LIN {X 0,Y 314.031,Z 449.566,A -85,B 0,C 180,E1 -15906.575,E2 -15906.575} C_VEL
LIN {X 0,Y 314.681,Z 456.551,A -85,B 0,C 180,E1 -15906.784,E2 -15906.784} C_VEL
LIN {X 0,Y 313.281,Z 518.504,A -85,B 0,C 180,E1 -15908.189,E2 -15908.189} C_VEL
LIN {X 0,Y 312.768,Z 530.956,A -85,B 0,C 180,E1 -15908.671,E2 -15908.671} C_VEL
LIN {X 0,Y 311.794,Z 543.197,A -85,B 0,C 180,E1 -15909.379,E2 -15909.379} C_VEL
LIN {X 0,Y 310.634,Z 555.216,A -85,B 0,C 180,E1 -15910.334,E2 -15910.334} C_VEL
LIN {X 0,Y 309.413,Z 566.12,A -85,B 0,C 180,E1 -15911.459,E2 -15911.459} C_VEL
LIN {X 0,Y 308.122,Z 576.138,A -85,B 0,C 180,E1 -15912.752,E2 -15912.752} C_VEL
LIN {X 0,Y 307.026,Z 586.271,A -85,B 0,C 180,E1 -15914.398,E2 -15914.398} C_VEL
LIN {X 0,Y 305.821,Z 596.058,A -85,B 0,C 180,E1 -15916.376,E2 -15916.376} C_VEL
LIN {X 0,Y 304.804,Z 603.833,A -85,B 0,C 180,E1 -15918.361,E2 -15918.361} C_VEL
LIN {X 0,Y 304.154,Z 610.997,A -85,B 0,C 180,E1 -15920.692,E2 -15920.692} C_VEL
LIN {X 0,Y 303.824,Z 615.751,A -85,B 0,C 180,E1 -15922.691,E2 -15922.691} C_VEL
LIN {X 0,Y 303.696,Z 619.372,A -85,B 0,C 180,E1 -15924.689,E2 -15924.689} C_VEL
LIN {X 0,Y 303.709,Z 621.23,A -85,B 0,C 180,E1 -15926.019,E2 -15926.019} C_VEL
LIN {X 0,Y 303.691,Z 622.612,A -85,B 0,C 180,E1 -15927.347,E2 -15927.347} C_VEL
LIN {X 0,Y 303.723,Z 623.593,A -85,B 0,C 180,E1 -15928.674,E2 -15928.674} C_VEL
LIN {X 0,Y 303.764,Z 624.179,A -85,B 0,C 180,E1 -15930,E2 -15930} C_VEL
LIN {X 0,Y 303.684,Z 624.356,A -85,B 0,C 180,E1 -15931.326,E2 -15931.326} C_VEL
LIN {X 0,Y 303.657,Z 624.102,A -85,B 0,C 180,E1 -15932.653,E2 -15932.653} C_VEL
LIN {X 0,Y 303.66,Z 623.46,A -85,B 0,C 180,E1 -15933.981,E2 -15933.981} C_VEL
LIN {X 0,Y 303.659,Z 622.155,A -85,B 0,C 180,E1 -15935.611,E2 -15935.611} C_VEL
LIN {X 0,Y 303.947,Z 619.106,A -85,B 0,C 180,E1 -15937.974,E2 -15937.974} C_VEL
LIN {X 0,Y 304.415,Z 615.463,A -85,B 0,C 180,E1 -15939.971,E2 -15939.971} C_VEL
LIN {X 0,Y 305.165,Z 610.729,A -85,B 0,C 180,E1 -15941.962,E2 -15941.962} C_VEL
LIN {X 0,Y 306.656,Z 603.648,A -85,B 0,C 180,E1 -15944.263,E2 -15944.263} C_VEL
LIN {X 0,Y 308.039,Z 596.351,A -85,B 0,C 180,E1 -15946.143,E2 -15946.143} C_VEL
LIN {X 0,Y 309.559,Z 588.201,A -85,B 0,C 180,E1 -15947.848,E2 -15947.848} C_VEL
LIN {X 0,Y 311.381,Z 578.704,A -85,B 0,C 180,E1 -15949.445,E2 -15949.445} C_VEL
LIN {X 0,Y 313.312,Z 568.196,A -85,B 0,C 180,E1 -15950.86,E2 -15950.86} C_VEL
LIN {X 0,Y 315.192,Z 556.51,A -85,B 0,C 180,E1 -15952.102,E2 -15952.102} C_VEL
LIN {X 0,Y 316.76,Z 545.154,A -85,B 0,C 180,E1 -15953.019,E2 -15953.019} C_VEL
LIN {X 0,Y 318.203,Z 531.649,A -85,B 0,C 180,E1 -15953.813,E2 -15953.813} C_VEL
LIN {X 0,Y 319.058,Z 519.098,A -85,B 0,C 180,E1 -15954.307,E2 -15954.307} C_VEL
LIN {X 0,Y 320.823,Z 456.805,A -85,B 0,C 180,E1 -15955.725,E2 -15955.725} C_VEL
LIN {X 0,Y 317.597,Z 436.667,A -85,B 0,C 180,E1 -15956.559,E2 -15956.559} C_VEL
LIN {X 0,Y 313.376,Z 415.766,A -85,B 0,C 180,E1 -15957.545,E2 -15957.545} C_VEL
LIN {X 0,Y 311.73,Z 410.591,A -85,B 0,C 180,E1 -15957.875,E2 -15957.875} C_VEL
LIN {X 0,Y 309.758,Z 401.062,A -85,B 0,C 180,E1 -15960.871,E2 -15960.871} C_VEL
LIN {X 0,Y 307.599,Z 391.784,A -85,B 0,C 180,E1 -15963.953,E2 -15963.953} C_VEL
LIN {X 0,Y 305.496,Z 383.432,A -85,B 0,C 180,E1 -15966.941,E2 -15966.941} C_VEL
LIN {X 0,Y 305.452,Z 383.433,A -85,B 0,C 180,E1 -15970.599,E2 -15970.599} C_VEL
LIN {X 0,Y 305.451,Z 383.431,A -85,B 0,C 180,E1 -15974.499,E2 -15974.499} C_VEL
LIN {X 0,Y 305.492,Z 383.426,A -85,B 0,C 180,E1 -15978.152,E2 -15978.152} C_VEL
LIN {X 0,Y 305.515,Z 383.425,A -85,B 0,C 180,E1 -15981.604,E2 -15981.604} C_VEL
LIN {X 0,Y 305.457,Z 383.433,A -85,B 0,C 180,E1 -15984.886,E2 -15984.886} C_VEL
LIN {X 0,Y 305.446,Z 383.436,A -85,B 0,C 180,E1 -15988.355,E2 -15988.355} C_VEL
LIN {X 0,Y 305.515,Z 383.428,A -85,B 0,C 180,E1 -15991.113,E2 -15991.113} C_VEL
LIN {X 0,Y 305.565,Z 383.4,A -85,B 0,C 180,E1 -15994.088,E2 -15994.088} C_VEL
LIN {X 0,Y 305.494,Z 383.43,A -85,B 0,C 180,E1 -15998.403,E2 -15998.403} C_VEL
LIN {X 0,Y 305.584,Z 383.414,A -85,B 0,C 180,E1 -16001.217,E2 -16001.217} C_VEL
LIN {X 0,Y 305.642,Z 383.406,A -85,B 0,C 180,E1 -16005.349,E2 -16005.349} C_VEL
LIN {X 0,Y 305.634,Z 383.406,A -85,B 0,C 180,E1 -16009.4,E2 -16009.4} C_VEL
LIN {X 0,Y 305.806,Z 383.391,A -85,B 0,C 180,E1 -16012.074,E2 -16012.074} C_VEL
LIN {X 0,Y 305.684,Z 383.399,A -85,B 0,C 180,E1 -16014.724,E2 -16014.724} C_VEL
LIN {X 0,Y 305.952,Z 383.366,A -85,B 0,C 180,E1 -16018.684,E2 -16018.684} C_VEL
LIN {X 0,Y 305.952,Z 383.374,A -85,B 0,C 180,E1 -16021.317,E2 -16021.317} C_VEL
LIN {X 0,Y 305.682,Z 383.408,A -85,B 0,C 180,E1 -16025.277,E2 -16025.277} C_VEL
LIN {X 0,Y 305.791,Z 383.386,A -85,B 0,C 180,E1 -16027.927,E2 -16027.927} C_VEL
LIN {X 0,Y 305.597,Z 383.414,A -85,B 0,C 180,E1 -16031.946,E2 -16031.946} C_VEL
LIN {X 0,Y 305.632,Z 383.414,A -85,B 0,C 180,E1 -16035.035,E2 -16035.035} C_VEL
LIN {X 0,Y 305.572,Z 383.42,A -85,B 0,C 180,E1 -16039.446,E2 -16039.446} C_VEL
LIN {X 0,Y 305.485,Z 383.432,A -85,B 0,C 180,E1 -16043.042,E2 -16043.042} C_VEL
LIN {X 0,Y 305.522,Z 383.403,A -85,B 0,C 180,E1 -16046.22,E2 -16046.22} C_VEL
LIN {X 0,Y 305.492,Z 383.431,A -85,B 0,C 180,E1 -16049.051,E2 -16049.051} C_VEL
LIN {X 0,Y 305.462,Z 383.435,A -85,B 0,C 180,E1 -16053.518,E2 -16053.518} C_VEL
LIN {X 0,Y 305.5,Z 383.429,A -85,B 0,C 180,E1 -16056.737,E2 -16056.737} C_VEL
LIN {X 0,Y 305.483,Z 383.437,A -85,B 0,C 180,E1 -16060.608,E2 -16060.608} C_VEL
LIN {X 0,Y 305.495,Z 383.433,A -85,B 0,C 180,E1 -16063.643,E2 -16063.643} C_VEL
LIN {X 0,Y 305.498,Z 383.436,A -85,B 0,C 180,E1 -16067.406,E2 -16067.406} C_VEL
LIN {X 0,Y 305.499,Z 383.524,A -85,B 0,C 180,E1 -16071.315,E2 -16071.315} C_VEL
LIN {X 0,Y 306.248,Z 386.681,A -85,B 0,C 180,E1 -16072.562,E2 -16072.562} C_VEL
LIN {X 0,Y 315.185,Z 404.698,A -85,B 0,C 180,E1 -16074.052,E2 -16074.052} C_VEL
LIN {X 0,Y 321.757,Z 419.845,A -85,B 0,C 180,E1 -16075.128,E2 -16075.128} C_VEL
LIN {X 0,Y 319.665,Z 493.003,A -85,B 0,C 180,E1 -16076.799,E2 -16076.799} C_VEL
LIN {X 0,Y 318.957,Z 504.93,A -85,B 0,C 180,E1 -16077.286,E2 -16077.286} C_VEL
LIN {X 0,Y 317.868,Z 517.514,A -85,B 0,C 180,E1 -16078.046,E2 -16078.046} C_VEL
LIN {X 0,Y 316.481,Z 528.377,A -85,B 0,C 180,E1 -16078.916,E2 -16078.916} C_VEL
LIN {X 0,Y 315.108,Z 539.273,A -85,B 0,C 180,E1 -16080.064,E2 -16080.064} C_VEL
LIN {X 0,Y 313.649,Z 548.685,A -85,B 0,C 180,E1 -16081.297,E2 -16081.297} C_VEL
LIN {X 0,Y 311.819,Z 558.321,A -85,B 0,C 180,E1 -16082.845,E2 -16082.845} C_VEL
LIN {X 0,Y 309.966,Z 567.861,A -85,B 0,C 180,E1 -16084.772,E2 -16084.772} C_VEL
LIN {X 0,Y 308.261,Z 575.922,A -85,B 0,C 180,E1 -16086.842,E2 -16086.842} C_VEL
LIN {X 0,Y 307.062,Z 581.197,A -85,B 0,C 180,E1 -16088.519,E2 -16088.519} C_VEL
LIN {X 0,Y 306.066,Z 585.733,A -85,B 0,C 180,E1 -16090.3,E2 -16090.3} C_VEL
LIN {X 0,Y 305.073,Z 590.158,A -85,B 0,C 180,E1 -16092.574,E2 -16092.574} C_VEL
LIN {X 0,Y 304.649,Z 592.146,A -85,B 0,C 180,E1 -16093.929,E2 -16093.929} C_VEL
LIN {X 0,Y 304.192,Z 594.355,A -85,B 0,C 180,E1 -16096.019,E2 -16096.019} C_VEL
LIN {X 0,Y 303.847,Z 595.527,A -85,B 0,C 180,E1 -16097.985,E2 -16097.985} C_VEL
LIN {X 0,Y 303.635,Z 595.748,A -85,B 0,C 180,E1 -16100.676,E2 -16100.676} C_VEL
LIN {X 0,Y 303.703,Z 595.242,A -85,B 0,C 180,E1 -16102.019,E2 -16102.019} C_VEL
LIN {X 0,Y 303.858,Z 593.743,A -85,B 0,C 180,E1 -16104.026,E2 -16104.026} C_VEL
LIN {X 0,Y 304.04,Z 590.269,A -85,B 0,C 180,E1 -16106.687,E2 -16106.687} C_VEL
LIN {X 0,Y 304.454,Z 586.504,A -85,B 0,C 180,E1 -16108.677,E2 -16108.677} C_VEL
LIN {X 0,Y 304.913,Z 581.638,A -85,B 0,C 180,E1 -16110.66,E2 -16110.66} C_VEL
LIN {X 0,Y 305.744,Z 575.501,A -85,B 0,C 180,E1 -16112.635,E2 -16112.635} C_VEL
LIN {X 0,Y 306.819,Z 567.863,A -85,B 0,C 180,E1 -16114.598,E2 -16114.598} C_VEL
LIN {X 0,Y 307.989,Z 558.298,A -85,B 0,C 180,E1 -16116.551,E2 -16116.551} C_VEL
LIN {X 0,Y 309.298,Z 548.412,A -85,B 0,C 180,E1 -16118.164,E2 -16118.164} C_VEL
LIN {X 0,Y 310.604,Z 537.252,A -85,B 0,C 180,E1 -16119.606,E2 -16119.606} C_VEL
LIN {X 0,Y 311.597,Z 526.36,A -85,B 0,C 180,E1 -16120.724,E2 -16120.724} C_VEL
LIN {X 0,Y 312.452,Z 515.426,A -85,B 0,C 180,E1 -16121.597,E2 -16121.597} C_VEL
LIN {X 0,Y 313.24,Z 502.643,A -85,B 0,C 180,E1 -16122.348,E2 -16122.348} C_VEL
LIN {X 0,Y 313.687,Z 490.148,A -85,B 0,C 180,E1 -16122.823,E2 -16122.823} C_VEL
LIN {X 0,Y 315.394,Z 413.357,A -85,B 0,C 180,E1 -16124.561,E2 -16124.561} C_VEL
LIN {X 0,Y 313.375,Z 405.881,A -85,B 0,C 180,E1 -16124.88,E2 -16124.88} C_VEL
LIN {X 0,Y 306.036,Z 385.635,A -85,B 0,C 180,E1 -16125.931,E2 -16125.931} C_VEL
LIN {X 0,Y 305.595,Z 383.422,A -85,B 0,C 180,E1 -16126.706,E2 -16126.706} C_VEL
LIN {X 0,Y 305.524,Z 383.429,A -85,B 0,C 180,E1 -16130.184,E2 -16130.184} C_VEL
LIN {X 0,Y 305.511,Z 383.428,A -85,B 0,C 180,E1 -16134.46,E2 -16134.46} C_VEL
LIN {X 0,Y 305.543,Z 383.423,A -85,B 0,C 180,E1 -16137.389,E2 -16137.389} C_VEL
LIN {X 0,Y 305.468,Z 383.437,A -85,B 0,C 180,E1 -16140.408,E2 -16140.408} C_VEL
LIN {X 0,Y 305.466,Z 383.435,A -85,B 0,C 180,E1 -16144.077,E2 -16144.077} C_VEL
LIN {X 0,Y 305.475,Z 383.433,A -85,B 0,C 180,E1 -16146.738,E2 -16146.738} C_VEL
LIN {X 0,Y 305.454,Z 383.433,A -85,B 0,C 180,E1 -16150.599,E2 -16150.599} C_VEL
LIN {X 0,Y 305.461,Z 383.435,A -85,B 0,C 180,E1 -16154.5,E2 -16154.5} C_VEL
LIN {X 0,Y 305.495,Z 383.427,A -85,B 0,C 180,E1 -16158.151,E2 -16158.151} C_VEL
LIN {X 0,Y 305.476,Z 383.427,A -85,B 0,C 180,E1 -16158.771,E2 -16158.771} C_VEL
LIN {X 0,Y 304.812,Z 383.515,A -85,B 0,C 180,E1 -16159.872,E2 -16159.872} C_VEL
LIN {X 0,Y 301.957,Z 383.87,A -85,B 0,C 180,E1 -16161.665,E2 -16161.665} C_VEL
LIN {X 0,Y 299.53,Z 384.171,A -85,B 0,C 180,E1 -16163.118,E2 -16163.118} C_VEL
LIN {X 0,Y 298.487,Z 384.3,A -85,B 0,C 180,E1 -16164.244,E2 -16164.244} C_VEL
LIN {X 0,Y 298.401,Z 384.306,A -85,B 0,C 180,E1 -16164.626,E2 -16164.626} C_VEL
LIN {X 0,Y 298.388,Z 384.315,A -85,B 0,C 180,E1 -16168.79,E2 -16168.79} C_VEL
LIN {X 0,Y 298.454,Z 384.307,A -85,B 0,C 180,E1 -16171.903,E2 -16171.903} C_VEL
LIN {X 0,Y 298.481,Z 384.297,A -85,B 0,C 180,E1 -16174.923,E2 -16174.923} C_VEL
LIN {X 0,Y 298.46,Z 384.305,A -85,B 0,C 180,E1 -16179.316,E2 -16179.316} C_VEL
LIN {X 0,Y 298.533,Z 384.296,A -85,B 0,C 180,E1 -16182.179,E2 -16182.179} C_VEL
LIN {X 0,Y 298.587,Z 384.282,A -85,B 0,C 180,E1 -16184.994,E2 -16184.994} C_VEL
LIN {X 0,Y 298.589,Z 384.288,A -85,B 0,C 180,E1 -16189.146,E2 -16189.146} C_VEL
LIN {X 0,Y 298.752,Z 384.27,A -85,B 0,C 180,E1 -16191.885,E2 -16191.885} C_VEL
LIN {X 0,Y 298.654,Z 384.273,A -85,B 0,C 180,E1 -16194.598,E2 -16194.598} C_VEL
LIN {X 0,Y 298.919,Z 384.248,A -85,B 0,C 180,E1 -16198.652,E2 -16198.652} C_VEL
LIN {X 0,Y 298.919,Z 384.248,A -85,B 0,C 180,E1 -16201.347,E2 -16201.347} C_VEL
LIN {X 0,Y 298.791,Z 384.264,A -85,B 0,C 180,E1 -16206.754,E2 -16206.754} C_VEL
LIN {X 0,Y 298.675,Z 384.278,A -85,B 0,C 180,E1 -16209.48,E2 -16209.48} C_VEL
LIN {X 0,Y 298.547,Z 384.295,A -85,B 0,C 180,E1 -16213.615,E2 -16213.615} C_VEL
LIN {X 0,Y 298.542,Z 384.297,A -85,B 0,C 180,E1 -16216.409,E2 -16216.409} C_VEL
LIN {X 0,Y 298.51,Z 384.299,A -85,B 0,C 180,E1 -16219.657,E2 -16219.657} C_VEL
LIN {X 0,Y 298.452,Z 384.307,A -85,B 0,C 180,E1 -16223.598,E2 -16223.598} C_VEL
LIN {X 0,Y 298.481,Z 384.303,A -85,B 0,C 180,E1 -16226.575,E2 -16226.575} C_VEL
LIN {X 0,Y 298.411,Z 384.314,A -85,B 0,C 180,E1 -16229.642,E2 -16229.642} C_VEL
LIN {X 0,Y 298.39,Z 384.314,A -85,B 0,C 180,E1 -16232.801,E2 -16232.801} C_VEL
LIN {X 0,Y 298.465,Z 384.305,A -85,B 0,C 180,E1 -16236.814,E2 -16236.814} C_VEL
LIN {X 0,Y 298.451,Z 384.307,A -85,B 0,C 180,E1 -16241.103,E2 -16241.103} C_VEL
LIN {X 0,Y 298.455,Z 384.306,A -85,B 0,C 180,E1 -16243.116,E2 -16243.116} C_VEL
LIN {X 0,Y 298.429,Z 384.309,A -85,B 0,C 180,E1 -16246.927,E2 -16246.927} C_VEL
LIN {X 0,Y 298.412,Z 384.312,A -85,B 0,C 180,E1 -16251.004,E2 -16251.004} C_VEL
LIN {X 0,Y 298.43,Z 384.313,A -85,B 0,C 180,E1 -16253.933,E2 -16253.933} C_VEL
LIN {X 0,Y 298.472,Z 384.46,A -85,B 0,C 180,E1 -16256.959,E2 -16256.959} C_VEL
LIN {X 0,Y 300.719,Z 394.722,A -85,B 0,C 180,E1 -16260.125,E2 -16260.125} C_VEL
LIN {X 0,Y 302.598,Z 404.683,A -85,B 0,C 180,E1 -16263.071,E2 -16263.071} C_VEL
LIN {X 0,Y 302.438,Z 408.558,A -85,B 0,C 180,E1 -16264.133,E2 -16264.133} C_VEL
LIN {X 0,Y 302.109,Z 410.992,A -85,B 0,C 180,E1 -16264.783,E2 -16264.783} C_VEL
LIN {X 0,Y 307.048,Z 447.973,A -85,B 0,C 180,E1 -16266.067,E2 -16266.067} C_VEL
LIN {X 0,Y 308.01,Z 456.583,A -85,B 0,C 180,E1 -16266.343,E2 -16266.343} C_VEL
LIN {X 0,Y 306.567,Z 518.379,A -85,B 0,C 180,E1 -16267.775,E2 -16267.775} C_VEL
LIN {X 0,Y 305.972,Z 531.497,A -85,B 0,C 180,E1 -16268.306,E2 -16268.306} C_VEL
LIN {X 0,Y 304.915,Z 544.079,A -85,B 0,C 180,E1 -16269.068,E2 -16269.068} C_VEL
LIN {X 0,Y 303.741,Z 555.836,A -85,B 0,C 180,E1 -16270.045,E2 -16270.045} C_VEL
LIN {X 0,Y 302.476,Z 566.54,A -85,B 0,C 180,E1 -16271.193,E2 -16271.193} C_VEL
LIN {X 0,Y 301.148,Z 576.39,A -85,B 0,C 180,E1 -16272.515,E2 -16272.515} C_VEL
LIN {X 0,Y 300.032,Z 586.208,A -85,B 0,C 180,E1 -16274.158,E2 -16274.158} C_VEL
LIN {X 0,Y 298.863,Z 595.373,A -85,B 0,C 180,E1 -16276.053,E2 -16276.053} C_VEL
LIN {X 0,Y 297.819,Z 603.237,A -85,B 0,C 180,E1 -16278.084,E2 -16278.084} C_VEL
LIN {X 0,Y 297.101,Z 610.45,A -85,B 0,C 180,E1 -16280.469,E2 -16280.469} C_VEL
LIN {X 0,Y 296.772,Z 615.252,A -85,B 0,C 180,E1 -16282.516,E2 -16282.516} C_VEL
LIN {X 0,Y 296.62,Z 618.915,A -85,B 0,C 180,E1 -16284.562,E2 -16284.562} C_VEL
LIN {X 0,Y 296.621,Z 620.803,A -85,B 0,C 180,E1 -16285.924,E2 -16285.924} C_VEL
LIN {X 0,Y 296.613,Z 622.214,A -85,B 0,C 180,E1 -16287.284,E2 -16287.284} C_VEL
LIN {X 0,Y 296.634,Z 623.213,A -85,B 0,C 180,E1 -16288.642,E2 -16288.642} C_VEL
LIN {X 0,Y 296.673,Z 623.818,A -85,B 0,C 180,E1 -16290,E2 -16290} C_VEL
LIN {X 0,Y 296.597,Z 624.023,A -85,B 0,C 180,E1 -16291.358,E2 -16291.358} C_VEL
LIN {X 0,Y 296.58,Z 623.796,A -85,B 0,C 180,E1 -16292.716,E2 -16292.716} C_VEL
LIN {X 0,Y 296.573,Z 623.172,A -85,B 0,C 180,E1 -16294.077,E2 -16294.077} C_VEL
LIN {X 0,Y 296.655,Z 620.753,A -85,B 0,C 180,E1 -16296.803,E2 -16296.803} C_VEL
LIN {X 0,Y 297.04,Z 617.811,A -85,B 0,C 180,E1 -16298.846,E2 -16298.846} C_VEL
LIN {X 0,Y 297.653,Z 613.853,A -85,B 0,C 180,E1 -16300.888,E2 -16300.888} C_VEL
LIN {X 0,Y 298.574,Z 608.782,A -85,B 0,C 180,E1 -16302.921,E2 -16302.921} C_VEL
LIN {X 0,Y 300.015,Z 602.442,A -85,B 0,C 180,E1 -16304.932,E2 -16304.932} C_VEL
LIN {X 0,Y 301.657,Z 594.115,A -85,B 0,C 180,E1 -16307.028,E2 -16307.028} C_VEL
LIN {X 0,Y 303.52,Z 584.719,A -85,B 0,C 180,E1 -16308.915,E2 -16308.915} C_VEL
LIN {X 0,Y 305.601,Z 574.521,A -85,B 0,C 180,E1 -16310.53,E2 -16310.53} C_VEL
LIN {X 0,Y 307.633,Z 563.029,A -85,B 0,C 180,E1 -16311.968,E2 -16311.968} C_VEL
LIN {X 0,Y 309.397,Z 551.737,A -85,B 0,C 180,E1 -16313.068,E2 -16313.068} C_VEL
LIN {X 0,Y 310.971,Z 540.209,A -85,B 0,C 180,E1 -16313.915,E2 -16313.915} C_VEL
LIN {X 0,Y 312.231,Z 527.003,A -85,B 0,C 180,E1 -16314.608,E2 -16314.608} C_VEL
LIN {X 0,Y 313.046,Z 514.207,A -85,B 0,C 180,E1 -16315.027,E2 -16315.027} C_VEL
LIN {X 0,Y 314.597,Z 457.765,A -85,B 0,C 180,E1 -16316.325,E2 -16316.325} C_VEL
LIN {X 0,Y 311.364,Z 437.492,A -85,B 0,C 180,E1 -16317.193,E2 -16317.193} C_VEL
LIN {X 0,Y 307.278,Z 417.254,A -85,B 0,C 180,E1 -16318.181,E2 -16318.181} C_VEL
LIN {X 0,Y 304.522,Z 410.161,A -85,B 0,C 180,E1 -16318.718,E2 -16318.718} C_VEL
LIN {X 0,Y 302.101,Z 399.117,A -85,B 0,C 180,E1 -16322.348,E2 -16322.348} C_VEL
LIN {X 0,Y 299.654,Z 389.019,A -85,B 0,C 180,E1 -16325.897,E2 -16325.897} C_VEL
LIN {X 0,Y 298.473,Z 384.306,A -85,B 0,C 180,E1 -16327.683,E2 -16327.683} C_VEL
LIN {X 0,Y 298.383,Z 384.314,A -85,B 0,C 180,E1 -16331.261,E2 -16331.261} C_VEL
LIN {X 0,Y 298.413,Z 384.308,A -85,B 0,C 180,E1 -16335.046,E2 -16335.046} C_VEL
LIN {X 0,Y 298.451,Z 384.302,A -85,B 0,C 180,E1 -16338.75,E2 -16338.75} C_VEL
LIN {X 0,Y 298.443,Z 384.305,A -85,B 0,C 180,E1 -16342.246,E2 -16342.246} C_VEL
LIN {X 0,Y 298.403,Z 384.314,A -85,B 0,C 180,E1 -16345.581,E2 -16345.581} C_VEL
LIN {X 0,Y 298.39,Z 384.316,A -85,B 0,C 180,E1 -16348.791,E2 -16348.791} C_VEL
LIN {X 0,Y 298.458,Z 384.307,A -85,B 0,C 180,E1 -16351.904,E2 -16351.904} C_VEL
LIN {X 0,Y 298.479,Z 384.277,A -85,B 0,C 180,E1 -16354.924,E2 -16354.924} C_VEL
LIN {X 0,Y 298.444,Z 384.309,A -85,B 0,C 180,E1 -16359.315,E2 -16359.315} C_VEL
LIN {X 0,Y 298.531,Z 384.296,A -85,B 0,C 180,E1 -16362.179,E2 -16362.179} C_VEL
LIN {X 0,Y 298.587,Z 384.284,A -85,B 0,C 180,E1 -16364.995,E2 -16364.995} C_VEL
LIN {X 0,Y 298.589,Z 384.284,A -85,B 0,C 180,E1 -16369.147,E2 -16369.147} C_VEL
LIN {X 0,Y 298.751,Z 384.27,A -85,B 0,C 180,E1 -16371.886,E2 -16371.886} C_VEL
LIN {X 0,Y 298.655,Z 384.274,A -85,B 0,C 180,E1 -16374.599,E2 -16374.599} C_VEL
LIN {X 0,Y 298.919,Z 384.242,A -85,B 0,C 180,E1 -16378.653,E2 -16378.653} C_VEL
LIN {X 0,Y 298.919,Z 384.25,A -85,B 0,C 180,E1 -16381.348,E2 -16381.348} C_VEL
LIN {X 0,Y 298.781,Z 384.265,A -85,B 0,C 180,E1 -16386.755,E2 -16386.755} C_VEL
LIN {X 0,Y 298.629,Z 384.284,A -85,B 0,C 180,E1 -16389.483,E2 -16389.483} C_VEL
LIN {X 0,Y 298.546,Z 384.293,A -85,B 0,C 180,E1 -16393.616,E2 -16393.616} C_VEL
LIN {X 0,Y 298.543,Z 384.292,A -85,B 0,C 180,E1 -16396.409,E2 -16396.409} C_VEL
LIN {X 0,Y 298.507,Z 384.301,A -85,B 0,C 180,E1 -16399.655,E2 -16399.655} C_VEL
LIN {X 0,Y 298.453,Z 384.307,A -85,B 0,C 180,E1 -16403.599,E2 -16403.599} C_VEL
LIN {X 0,Y 298.481,Z 384.279,A -85,B 0,C 180,E1 -16406.576,E2 -16406.576} C_VEL
LIN {X 0,Y 298.417,Z 384.313,A -85,B 0,C 180,E1 -16409.642,E2 -16409.642} C_VEL
LIN {X 0,Y 298.392,Z 384.316,A -85,B 0,C 180,E1 -16412.801,E2 -16412.801} C_VEL
LIN {X 0,Y 298.468,Z 384.305,A -85,B 0,C 180,E1 -16416.815,E2 -16416.815} C_VEL
LIN {X 0,Y 298.45,Z 384.31,A -85,B 0,C 180,E1 -16421.251,E2 -16421.251} C_VEL
LIN {X 0,Y 298.417,Z 384.319,A -85,B 0,C 180,E1 -16425.048,E2 -16425.048} C_VEL
LIN {X 0,Y 298.42,Z 384.318,A -85,B 0,C 180,E1 -16428.746,E2 -16428.746} C_VEL
LIN {X 0,Y 298.442,Z 384.336,A -85,B 0,C 180,E1 -16430.593,E2 -16430.593} C_VEL
LIN {X 0,Y 299.127,Z 387.198,A -85,B 0,C 180,E1 -16431.71,E2 -16431.71} C_VEL
LIN {X 0,Y 308.479,Z 405.641,A -85,B 0,C 180,E1 -16433.333,E2 -16433.333} C_VEL
LIN {X 0,Y 315.617,Z 421.901,A -85,B 0,C 180,E1 -16434.544,E2 -16434.544} C_VEL
LIN {X 0,Y 313.411,Z 493.482,A -85,B 0,C 180,E1 -16436.204,E2 -16436.204} C_VEL
LIN {X 0,Y 312.64,Z 505.613,A -85,B 0,C 180,E1 -16436.711,E2 -16436.711} C_VEL
LIN {X 0,Y 311.491,Z 518.351,A -85,B 0,C 180,E1 -16437.503,E2 -16437.503} C_VEL
LIN {X 0,Y 310.045,Z 529.099,A -85,B 0,C 180,E1 -16438.387,E2 -16438.387} C_VEL
LIN {X 0,Y 308.6,Z 539.894,A -85,B 0,C 180,E1 -16439.555,E2 -16439.555} C_VEL
LIN {X 0,Y 306.869,Z 550.302,A -85,B 0,C 180,E1 -16440.971,E2 -16440.971} C_VEL
LIN {X 0,Y 304.992,Z 559.748,A -85,B 0,C 180,E1 -16442.558,E2 -16442.558} C_VEL
LIN {X 0,Y 303.095,Z 568.961,A -85,B 0,C 180,E1 -16444.497,E2 -16444.497} C_VEL
LIN {X 0,Y 301.294,Z 576.936,A -85,B 0,C 180,E1 -16446.638,E2 -16446.638} C_VEL
LIN {X 0,Y 299.845,Z 582.994,A -85,B 0,C 180,E1 -16448.697,E2 -16448.697} C_VEL
LIN {X 0,Y 298.742,Z 587.747,A -85,B 0,C 180,E1 -16450.771,E2 -16450.771} C_VEL
LIN {X 0,Y 297.913,Z 591.348,A -85,B 0,C 180,E1 -16452.85,E2 -16452.85} C_VEL
LIN {X 0,Y 297.318,Z 593.901,A -85,B 0,C 180,E1 -16454.929,E2 -16454.929} C_VEL
LIN {X 0,Y 297.053,Z 595.084,A -85,B 0,C 180,E1 -16456.315,E2 -16456.315} C_VEL
LIN {X 0,Y 296.821,Z 595.816,A -85,B 0,C 180,E1 -16457.696,E2 -16457.696} C_VEL
LIN {X 0,Y 296.541,Z 596.101,A -85,B 0,C 180,E1 -16460.451,E2 -16460.451} C_VEL
LIN {X 0,Y 296.606,Z 595.653,A -85,B 0,C 180,E1 -16461.827,E2 -16461.827} C_VEL
LIN {X 0,Y 296.765,Z 594.02,A -85,B 0,C 180,E1 -16464.074,E2 -16464.074} C_VEL
LIN {X 0,Y 296.946,Z 590.813,A -85,B 0,C 180,E1 -16466.608,E2 -16466.608} C_VEL
LIN {X 0,Y 297.375,Z 587.117,A -85,B 0,C 180,E1 -16468.646,E2 -16468.646} C_VEL
LIN {X 0,Y 297.836,Z 582.328,A -85,B 0,C 180,E1 -16470.676,E2 -16470.676} C_VEL
LIN {X 0,Y 298.671,Z 576.275,A -85,B 0,C 180,E1 -16472.697,E2 -16472.697} C_VEL
LIN {X 0,Y 299.766,Z 568.755,A -85,B 0,C 180,E1 -16474.707,E2 -16474.707} C_VEL
LIN {X 0,Y 300.757,Z 561.086,A -85,B 0,C 180,E1 -16476.373,E2 -16476.373} C_VEL
LIN {X 0,Y 302.145,Z 550.656,A -85,B 0,C 180,E1 -16478.191,E2 -16478.191} C_VEL
LIN {X 0,Y 303.46,Z 540.042,A -85,B 0,C 180,E1 -16479.666,E2 -16479.666} C_VEL
LIN {X 0,Y 304.53,Z 529.786,A -85,B 0,C 180,E1 -16480.807,E2 -16480.807} C_VEL
LIN {X 0,Y 305.535,Z 517.548,A -85,B 0,C 180,E1 -16481.863,E2 -16481.863} C_VEL
LIN {X 0,Y 306.434,Z 504.645,A -85,B 0,C 180,E1 -16482.668,E2 -16482.668} C_VEL
LIN {X 0,Y 306.928,Z 492.158,A -85,B 0,C 180,E1 -16483.195,E2 -16483.195} C_VEL
LIN {X 0,Y 308.756,Z 414.425,A -85,B 0,C 180,E1 -16484.997,E2 -16484.997} C_VEL
LIN {X 0,Y 305.841,Z 404.808,A -85,B 0,C 180,E1 -16485.445,E2 -16485.445} C_VEL
LIN {X 0,Y 298.882,Z 385.947,A -85,B 0,C 180,E1 -16486.477,E2 -16486.477} C_VEL
LIN {X 0,Y 298.535,Z 384.299,A -85,B 0,C 180,E1 -16487.113,E2 -16487.113} C_VEL
LIN {X 0,Y 298.455,Z 384.31,A -85,B 0,C 180,E1 -16490.684,E2 -16490.684} C_VEL
LIN {X 0,Y 298.489,Z 384.297,A -85,B 0,C 180,E1 -16495.075,E2 -16495.075} C_VEL
LIN {X 0,Y 298.478,Z 384.305,A -85,B 0,C 180,E1 -16498.093,E2 -16498.093} C_VEL
LIN {X 0,Y 298.397,Z 384.315,A -85,B 0,C 180,E1 -16502.799,E2 -16502.799} C_VEL
LIN {X 0,Y 298.447,Z 384.308,A -85,B 0,C 180,E1 -16506.807,E2 -16506.807} C_VEL
LIN {X 0,Y 298.409,Z 384.311,A -85,B 0,C 180,E1 -16509.485,E2 -16509.485} C_VEL
LIN {X 0,Y 298.425,Z 384.309,A -85,B 0,C 180,E1 -16513.108,E2 -16513.108} C_VEL
LIN {X 0,Y 298.466,Z 384.299,A -85,B 0,C 180,E1 -16516.931,E2 -16516.931} C_VEL
LIN {X 0,Y 298.438,Z 384.308,A -85,B 0,C 180,E1 -16520.997,E2 -16520.997} C_VEL
LIN {X 0,Y 298.401,Z 384.306,A -85,B 0,C 180,E1 -16524.626,E2 -16524.626} C_VEL
LIN {X 0,Y 297.734,Z 384.39,A -85,B 0,C 180,E1 -16525.752,E2 -16525.752} C_VEL
LIN {X 0,Y 294.897,Z 384.748,A -85,B 0,C 180,E1 -16527.585,E2 -16527.585} C_VEL
LIN {X 0,Y 292.49,Z 385.054,A -85,B 0,C 180,E1 -16529.073,E2 -16529.073} C_VEL
LIN {X 0,Y 291.455,Z 385.182,A -85,B 0,C 180,E1 -16530.225,E2 -16530.225} C_VEL
LIN {X 0,Y 291.368,Z 385.19,A -85,B 0,C 180,E1 -16530.616,E2 -16530.616} C_VEL
LIN {X 0,Y 291.41,Z 385.179,A -85,B 0,C 180,E1 -16534.271,E2 -16534.271} C_VEL
LIN {X 0,Y 291.385,Z 385.185,A -85,B 0,C 180,E1 -16537.299,E2 -16537.299} C_VEL
LIN {X 0,Y 291.458,Z 385.18,A -85,B 0,C 180,E1 -16540.27,E2 -16540.27} C_VEL
LIN {X 0,Y 291.535,Z 385.161,A -85,B 0,C 180,E1 -16544.634,E2 -16544.634} C_VEL
LIN {X 0,Y 291.533,Z 385.168,A -85,B 0,C 180,E1 -16548.88,E2 -16548.88} C_VEL
LIN {X 0,Y 291.703,Z 385.147,A -85,B 0,C 180,E1 -16551.688,E2 -16551.688} C_VEL
LIN {X 0,Y 291.625,Z 385.148,A -85,B 0,C 180,E1 -16554.468,E2 -16554.468} C_VEL
LIN {X 0,Y 291.885,Z 385.124,A -85,B 0,C 180,E1 -16558.62,E2 -16558.62} C_VEL
LIN {X 0,Y 291.885,Z 385.124,A -85,B 0,C 180,E1 -16561.379,E2 -16561.379} C_VEL
LIN {X 0,Y 291.74,Z 385.141,A -85,B 0,C 180,E1 -16566.918,E2 -16566.918} C_VEL
LIN {X 0,Y 291.623,Z 385.157,A -85,B 0,C 180,E1 -16569.712,E2 -16569.712} C_VEL
LIN {X 0,Y 291.516,Z 385.172,A -85,B 0,C 180,E1 -16573.95,E2 -16573.95} C_VEL
LIN {X 0,Y 291.481,Z 385.174,A -85,B 0,C 180,E1 -16576.818,E2 -16576.818} C_VEL
LIN {X 0,Y 291.446,Z 385.181,A -85,B 0,C 180,E1 -16579.875,E2 -16579.875} C_VEL
LIN {X 0,Y 291.394,Z 385.189,A -85,B 0,C 180,E1 -16584.206,E2 -16584.206} C_VEL
LIN {X 0,Y 291.414,Z 385.183,A -85,B 0,C 180,E1 -16587.272,E2 -16587.272} C_VEL
LIN {X 0,Y 291.328,Z 385.195,A -85,B 0,C 180,E1 -16590.438,E2 -16590.438} C_VEL
LIN {X 0,Y 291.339,Z 385.196,A -85,B 0,C 180,E1 -16593.699,E2 -16593.699} C_VEL
LIN {X 0,Y 291.4,Z 385.185,A -85,B 0,C 180,E1 -16597.262,E2 -16597.262} C_VEL
LIN {X 0,Y 291.401,Z 385.185,A -85,B 0,C 180,E1 -16600.631,E2 -16600.631} C_VEL
LIN {X 0,Y 291.349,Z 385.191,A -85,B 0,C 180,E1 -16604.39,E2 -16604.39} C_VEL
LIN {X 0,Y 291.35,Z 385.193,A -85,B 0,C 180,E1 -16608.399,E2 -16608.399} C_VEL
LIN {X 0,Y 291.362,Z 385.191,A -85,B 0,C 180,E1 -16611.161,E2 -16611.161} C_VEL
LIN {X 0,Y 291.383,Z 385.19,A -85,B 0,C 180,E1 -16614.63,E2 -16614.63} C_VEL
LIN {X 0,Y 291.431,Z 385.378,A -85,B 0,C 180,E1 -16616.545,E2 -16616.545} C_VEL
LIN {X 0,Y 293.965,Z 397.107,A -85,B 0,C 180,E1 -16620.26,E2 -16620.26} C_VEL
LIN {X 0,Y 295.562,Z 405.409,A -85,B 0,C 180,E1 -16622.776,E2 -16622.776} C_VEL
LIN {X 0,Y 295.707,Z 408.051,A -85,B 0,C 180,E1 -16623.537,E2 -16623.537} C_VEL
LIN {X 0,Y 295.332,Z 410.69,A -85,B 0,C 180,E1 -16624.259,E2 -16624.259} C_VEL
LIN {X 0,Y 300.207,Z 447.289,A -85,B 0,C 180,E1 -16625.567,E2 -16625.567} C_VEL
LIN {X 0,Y 301.35,Z 457.164,A -85,B 0,C 180,E1 -16625.896,E2 -16625.896} C_VEL
LIN {X 0,Y 299.869,Z 518.251,A -85,B 0,C 180,E1 -16627.342,E2 -16627.342} C_VEL
LIN {X 0,Y 299.248,Z 531.269,A -85,B 0,C 180,E1 -16627.883,E2 -16627.883} C_VEL
LIN {X 0,Y 298.157,Z 543.824,A -85,B 0,C 180,E1 -16628.662,E2 -16628.662} C_VEL
LIN {X 0,Y 296.854,Z 556.433,A -85,B 0,C 180,E1 -16629.743,E2 -16629.743} C_VEL
LIN {X 0,Y 295.327,Z 568.21,A -85,B 0,C 180,E1 -16631.081,E2 -16631.081} C_VEL
LIN {X 0,Y 293.914,Z 578.799,A -85,B 0,C 180,E1 -16632.609,E2 -16632.609} C_VEL
LIN {X 0,Y 292.942,Z 587.189,A -85,B 0,C 180,E1 -16634.108,E2 -16634.108} C_VEL
LIN {X 0,Y 291.741,Z 596.151,A -85,B 0,C 180,E1 -16636.061,E2 -16636.061} C_VEL
LIN {X 0,Y 290.68,Z 603.771,A -85,B 0,C 180,E1 -16638.141,E2 -16638.141} C_VEL
LIN {X 0,Y 290.065,Z 609.903,A -85,B 0,C 180,E1 -16640.235,E2 -16640.235} C_VEL
LIN {X 0,Y 289.7,Z 614.75,A -85,B 0,C 180,E1 -16642.332,E2 -16642.332} C_VEL
LIN {X 0,Y 289.556,Z 618.458,A -85,B 0,C 180,E1 -16644.429,E2 -16644.429} C_VEL
LIN {X 0,Y 289.537,Z 620.369,A -85,B 0,C 180,E1 -16645.824,E2 -16645.824} C_VEL
LIN {X 0,Y 289.538,Z 621.816,A -85,B 0,C 180,E1 -16647.217,E2 -16647.217} C_VEL
LIN {X 0,Y 289.548,Z 622.833,A -85,B 0,C 180,E1 -16648.609,E2 -16648.609} C_VEL
LIN {X 0,Y 289.583,Z 623.456,A -85,B 0,C 180,E1 -16650,E2 -16650} C_VEL
LIN {X 0,Y 289.512,Z 623.683,A -85,B 0,C 180,E1 -16651.391,E2 -16651.391} C_VEL
LIN {X 0,Y 289.505,Z 623.49,A -85,B 0,C 180,E1 -16652.783,E2 -16652.783} C_VEL
LIN {X 0,Y 289.48,Z 621.949,A -85,B 0,C 180,E1 -16655.499,E2 -16655.499} C_VEL
LIN {X 0,Y 289.581,Z 620.502,A -85,B 0,C 180,E1 -16656.97,E2 -16656.97} C_VEL
LIN {X 0,Y 290.006,Z 617.599,A -85,B 0,C 180,E1 -16659.063,E2 -16659.063} C_VEL
LIN {X 0,Y 290.643,Z 613.682,A -85,B 0,C 180,E1 -16661.154,E2 -16661.154} C_VEL
LIN {X 0,Y 291.639,Z 608.656,A -85,B 0,C 180,E1 -16663.234,E2 -16663.234} C_VEL
LIN {X 0,Y 293.128,Z 602.375,A -85,B 0,C 180,E1 -16665.291,E2 -16665.291} C_VEL
LIN {X 0,Y 294.754,Z 594.672,A -85,B 0,C 180,E1 -16667.31,E2 -16667.31} C_VEL
LIN {X 0,Y 296.411,Z 586.589,A -85,B 0,C 180,E1 -16669.027,E2 -16669.027} C_VEL
LIN {X 0,Y 298.513,Z 576.905,A -85,B 0,C 180,E1 -16670.68,E2 -16670.68} C_VEL
LIN {X 0,Y 300.639,Z 566.169,A -85,B 0,C 180,E1 -16672.144,E2 -16672.144} C_VEL
LIN {X 0,Y 302.456,Z 555.753,A -85,B 0,C 180,E1 -16673.267,E2 -16673.267} C_VEL
LIN {X 0,Y 304.104,Z 544.377,A -85,B 0,C 180,E1 -16674.218,E2 -16674.218} C_VEL
LIN {X 0,Y 305.543,Z 531.604,A -85,B 0,C 180,E1 -16675.002,E2 -16675.002} C_VEL
LIN {X 0,Y 306.569,Z 518.21,A -85,B 0,C 180,E1 -16675.548,E2 -16675.548} C_VEL
LIN {X 0,Y 308.41,Z 458.561,A -85,B 0,C 180,E1 -16676.955,E2 -16676.955} C_VEL
LIN {X 0,Y 305.24,Z 438.655,A -85,B 0,C 180,E1 -16677.835,E2 -16677.835} C_VEL
LIN {X 0,Y 301.365,Z 419.447,A -85,B 0,C 180,E1 -16678.807,E2 -16678.807} C_VEL
LIN {X 0,Y 298.357,Z 412.643,A -85,B 0,C 180,E1 -16679.359,E2 -16679.359} C_VEL
LIN {X 0,Y 297.245,Z 409.759,A -85,B 0,C 180,E1 -16679.603,E2 -16679.603} C_VEL
LIN {X 0,Y 294.921,Z 399.119,A -85,B 0,C 180,E1 -16683.235,E2 -16683.235} C_VEL
LIN {X 0,Y 292.384,Z 389.052,A -85,B 0,C 180,E1 -16686.935,E2 -16686.935} C_VEL
LIN {X 0,Y 291.372,Z 385.189,A -85,B 0,C 180,E1 -16688.432,E2 -16688.432} C_VEL
LIN {X 0,Y 291.337,Z 385.191,A -85,B 0,C 180,E1 -16692.488,E2 -16692.488} C_VEL
LIN {X 0,Y 291.367,Z 385.186,A -85,B 0,C 180,E1 -16696.353,E2 -16696.353} C_VEL
LIN {X 0,Y 291.409,Z 385.181,A -85,B 0,C 180,E1 -16700.51,E2 -16700.51} C_VEL
LIN {X 0,Y 291.429,Z 385.178,A -85,B 0,C 180,E1 -16702.923,E2 -16702.923} C_VEL
LIN {X 0,Y 291.34,Z 385.193,A -85,B 0,C 180,E1 -16706.301,E2 -16706.301} C_VEL
LIN {X 0,Y 291.382,Z 385.185,A -85,B 0,C 180,E1 -16710.26,E2 -16710.26} C_VEL
LIN {X 0,Y 291.41,Z 385.16,A -85,B 0,C 180,E1 -16714.272,E2 -16714.272} C_VEL
LIN {X 0,Y 291.376,Z 385.18,A -85,B 0,C 180,E1 -16717.299,E2 -16717.299} C_VEL
LIN {X 0,Y 291.452,Z 385.175,A -85,B 0,C 180,E1 -16720.27,E2 -16720.27} C_VEL
LIN {X 0,Y 291.534,Z 385.163,A -85,B 0,C 180,E1 -16724.634,E2 -16724.634} C_VEL
LIN {X 0,Y 291.532,Z 385.164,A -85,B 0,C 180,E1 -16728.881,E2 -16728.881} C_VEL
LIN {X 0,Y 291.702,Z 385.149,A -85,B 0,C 180,E1 -16731.689,E2 -16731.689} C_VEL
LIN {X 0,Y 291.625,Z 385.149,A -85,B 0,C 180,E1 -16734.469,E2 -16734.469} C_VEL
LIN {X 0,Y 291.885,Z 385.118,A -85,B 0,C 180,E1 -16738.621,E2 -16738.621} C_VEL
LIN {X 0,Y 291.885,Z 385.126,A -85,B 0,C 180,E1 -16741.38,E2 -16741.38} C_VEL
LIN {X 0,Y 291.73,Z 385.142,A -85,B 0,C 180,E1 -16746.919,E2 -16746.919} C_VEL
LIN {X 0,Y 291.569,Z 385.164,A -85,B 0,C 180,E1 -16749.714,E2 -16749.714} C_VEL
LIN {X 0,Y 291.516,Z 385.169,A -85,B 0,C 180,E1 -16753.951,E2 -16753.951} C_VEL
LIN {X 0,Y 291.481,Z 385.169,A -85,B 0,C 180,E1 -16756.819,E2 -16756.819} C_VEL
LIN {X 0,Y 291.446,Z 385.181,A -85,B 0,C 180,E1 -16759.876,E2 -16759.876} C_VEL
LIN {X 0,Y 291.395,Z 385.18,A -85,B 0,C 180,E1 -16764.206,E2 -16764.206} C_VEL
LIN {X 0,Y 291.416,Z 385.163,A -85,B 0,C 180,E1 -16767.273,E2 -16767.273} C_VEL
LIN {X 0,Y 291.334,Z 385.193,A -85,B 0,C 180,E1 -16770.438,E2 -16770.438} C_VEL
LIN {X 0,Y 291.342,Z 385.193,A -85,B 0,C 180,E1 -16773.699,E2 -16773.699} C_VEL
LIN {X 0,Y 291.402,Z 385.186,A -85,B 0,C 180,E1 -16777.262,E2 -16777.262} C_VEL
LIN {X 0,Y 291.4,Z 385.191,A -85,B 0,C 180,E1 -16780.632,E2 -16780.632} C_VEL
LIN {X 0,Y 291.354,Z 385.202,A -85,B 0,C 180,E1 -16784.391,E2 -16784.391} C_VEL
LIN {X 0,Y 291.357,Z 385.198,A -85,B 0,C 180,E1 -16788.399,E2 -16788.399} C_VEL
LIN {X 0,Y 291.386,Z 385.21,A -85,B 0,C 180,E1 -16789.843,E2 -16789.843} C_VEL
LIN {X 0,Y 291.934,Z 387.413,A -85,B 0,C 180,E1 -16790.787,E2 -16790.787} C_VEL
LIN {X 0,Y 302.028,Z 407.041,A -85,B 0,C 180,E1 -16792.619,E2 -16792.619} C_VEL
LIN {X 0,Y 309.465,Z 423.862,A -85,B 0,C 180,E1 -16793.93,E2 -16793.93} C_VEL
LIN {X 0,Y 307.186,Z 494.022,A -85,B 0,C 180,E1 -16795.587,E2 -16795.587} C_VEL
LIN {X 0,Y 306.348,Z 506.624,A -85,B 0,C 180,E1 -16796.132,E2 -16796.132} C_VEL
LIN {X 0,Y 305.135,Z 519.194,A -85,B 0,C 180,E1 -16796.937,E2 -16796.937} C_VEL
LIN {X 0,Y 303.396,Z 531.481,A -85,B 0,C 180,E1 -16798.003,E2 -16798.003} C_VEL
LIN {X 0,Y 301.696,Z 543.465,A -85,B 0,C 180,E1 -16799.41,E2 -16799.41} C_VEL
LIN {X 0,Y 299.755,Z 553.583,A -85,B 0,C 180,E1 -16800.89,E2 -16800.89} C_VEL
LIN {X 0,Y 297.835,Z 562.883,A -85,B 0,C 180,E1 -16802.605,E2 -16802.605} C_VEL
LIN {X 0,Y 295.835,Z 571.887,A -85,B 0,C 180,E1 -16804.684,E2 -16804.684} C_VEL
LIN {X 0,Y 294.08,Z 579.058,A -85,B 0,C 180,E1 -16806.777,E2 -16806.777} C_VEL
LIN {X 0,Y 292.636,Z 584.725,A -85,B 0,C 180,E1 -16808.885,E2 -16808.885} C_VEL
LIN {X 0,Y 291.558,Z 589.149,A -85,B 0,C 180,E1 -16811.01,E2 -16811.01} C_VEL
LIN {X 0,Y 290.727,Z 592.463,A -85,B 0,C 180,E1 -16813.137,E2 -16813.137} C_VEL
LIN {X 0,Y 290.083,Z 595.114,A -85,B 0,C 180,E1 -16815.723,E2 -16815.723} C_VEL
LIN {X 0,Y 289.769,Z 596.105,A -85,B 0,C 180,E1 -16817.392,E2 -16817.392} C_VEL
LIN {X 0,Y 289.465,Z 596.453,A -85,B 0,C 180,E1 -16820.215,E2 -16820.215} C_VEL
LIN {X 0,Y 289.504,Z 596.045,A -85,B 0,C 180,E1 -16821.625,E2 -16821.625} C_VEL
LIN {X 0,Y 289.677,Z 594.302,A -85,B 0,C 180,E1 -16824.117,E2 -16824.117} C_VEL
LIN {X 0,Y 289.856,Z 591.358,A -85,B 0,C 180,E1 -16826.525,E2 -16826.525} C_VEL
LIN {X 0,Y 290.297,Z 587.731,A -85,B 0,C 180,E1 -16828.613,E2 -16828.613} C_VEL
LIN {X 0,Y 290.763,Z 583.018,A -85,B 0,C 180,E1 -16830.692,E2 -16830.692} C_VEL
LIN {X 0,Y 291.768,Z 575.938,A -85,B 0,C 180,E1 -16833.107,E2 -16833.107} C_VEL
LIN {X 0,Y 292.919,Z 568.228,A -85,B 0,C 180,E1 -16835.162,E2 -16835.162} C_VEL
LIN {X 0,Y 294.228,Z 558.597,A -85,B 0,C 180,E1 -16837.204,E2 -16837.204} C_VEL
LIN {X 0,Y 295.635,Z 548.624,A -85,B 0,C 180,E1 -16838.889,E2 -16838.889} C_VEL
LIN {X 0,Y 297.044,Z 537.327,A -85,B 0,C 180,E1 -16840.393,E2 -16840.393} C_VEL
LIN {X 0,Y 298.111,Z 526.296,A -85,B 0,C 180,E1 -16841.559,E2 -16841.559} C_VEL
LIN {X 0,Y 299.05,Z 515.152,A -85,B 0,C 180,E1 -16842.469,E2 -16842.469} C_VEL
LIN {X 0,Y 299.839,Z 502.724,A -85,B 0,C 180,E1 -16843.21,E2 -16843.21} C_VEL
LIN {X 0,Y 300.34,Z 488.914,A -85,B 0,C 180,E1 -16843.731,E2 -16843.731} C_VEL
LIN {X 0,Y 302.067,Z 415.027,A -85,B 0,C 180,E1 -16845.468,E2 -16845.468} C_VEL
LIN {X 0,Y 295.46,Z 395.946,A -85,B 0,C 180,E1 -16846.462,E2 -16846.462} C_VEL
LIN {X 0,Y 291.708,Z 386.274,A -85,B 0,C 180,E1 -16847.048,E2 -16847.048} C_VEL
LIN {X 0,Y 291.509,Z 385.173,A -85,B 0,C 180,E1 -16847.538,E2 -16847.538} C_VEL
LIN {X 0,Y 291.381,Z 385.188,A -85,B 0,C 180,E1 -16851.21,E2 -16851.21} C_VEL
LIN {X 0,Y 291.403,Z 385.187,A -85,B 0,C 180,E1 -16854.204,E2 -16854.204} C_VEL
LIN {X 0,Y 291.439,Z 385.18,A -85,B 0,C 180,E1 -16857.269,E2 -16857.269} C_VEL
LIN {X 0,Y 291.341,Z 385.196,A -85,B 0,C 180,E1 -16860.436,E2 -16860.436} C_VEL
LIN {X 0,Y 291.346,Z 385.192,A -85,B 0,C 180,E1 -16863.697,E2 -16863.697} C_VEL
LIN {X 0,Y 291.382,Z 385.186,A -85,B 0,C 180,E1 -16867.254,E2 -16867.254} C_VEL
LIN {X 0,Y 291.334,Z 385.191,A -85,B 0,C 180,E1 -16870.641,E2 -16870.641} C_VEL
LIN {X 0,Y 291.342,Z 385.195,A -85,B 0,C 180,E1 -16874.391,E2 -16874.391} C_VEL
LIN {X 0,Y 291.387,Z 385.185,A -85,B 0,C 180,E1 -16878.389,E2 -16878.389} C_VEL
LIN {X 0,Y 291.386,Z 385.186,A -85,B 0,C 180,E1 -16881.163,E2 -16881.163} C_VEL
LIN {X 0,Y 291.384,Z 385.18,A -85,B 0,C 180,E1 -16884.629,E2 -16884.629} C_VEL
LIN {X 0,Y 291.367,Z 385.189,A -85,B 0,C 180,E1 -16887.949,E2 -16887.949} C_VEL
LIN {X 0,Y 291.368,Z 385.19,A -85,B 0,C 180,E1 -16890.616,E2 -16890.616} C_VEL
LIN {X 0,Y 290.714,Z 385.27,A -85,B 0,C 180,E1 -16891.769,E2 -16891.769} C_VEL
LIN {X 0,Y 287.928,Z 385.617,A -85,B 0,C 180,E1 -16893.648,E2 -16893.648} C_VEL
LIN {X 0,Y 285.537,Z 385.917,A -85,B 0,C 180,E1 -16895.173,E2 -16895.173} C_VEL
LIN {X 0,Y 284.47,Z 386.049,A -85,B 0,C 180,E1 -16896.353,E2 -16896.353} C_VEL
LIN {X 0,Y 284.361,Z 386.061,A -85,B 0,C 180,E1 -16896.753,E2 -16896.753} C_VEL
LIN {X 0,Y 284.401,Z 386.055,A -85,B 0,C 180,E1 -16901.261,E2 -16901.261} C_VEL
LIN {X 0,Y 284.473,Z 386.04,A -85,B 0,C 180,E1 -16904.469,E2 -16904.469} C_VEL
LIN {X 0,Y 284.484,Z 386.047,A -85,B 0,C 180,E1 -16908.601,E2 -16908.601} C_VEL
LIN {X 0,Y 284.653,Z 386.024,A -85,B 0,C 180,E1 -16911.481,E2 -16911.481} C_VEL
LIN {X 0,Y 284.595,Z 386.023,A -85,B 0,C 180,E1 -16914.331,E2 -16914.331} C_VEL
LIN {X 0,Y 284.851,Z 386.001,A -85,B 0,C 180,E1 -16918.586,E2 -16918.586} C_VEL
LIN {X 0,Y 284.851,Z 386,A -85,B 0,C 180,E1 -16921.413,E2 -16921.413} C_VEL
LIN {X 0,Y 284.692,Z 386.019,A -85,B 0,C 180,E1 -16927.09,E2 -16927.09} C_VEL
LIN {X 0,Y 284.561,Z 386.039,A -85,B 0,C 180,E1 -16929.955,E2 -16929.955} C_VEL
LIN {X 0,Y 284.472,Z 386.049,A -85,B 0,C 180,E1 -16934.303,E2 -16934.303} C_VEL
LIN {X 0,Y 284.42,Z 386.054,A -85,B 0,C 180,E1 -16937.248,E2 -16937.248} C_VEL
LIN {X 0,Y 284.375,Z 386.063,A -85,B 0,C 180,E1 -16940.242,E2 -16940.242} C_VEL
LIN {X 0,Y 284.363,Z 386.063,A -85,B 0,C 180,E1 -16943.875,E2 -16943.875} C_VEL
LIN {X 0,Y 284.39,Z 386.058,A -85,B 0,C 180,E1 -16947.173,E2 -16947.173} C_VEL
LIN {X 0,Y 284.288,Z 386.072,A -85,B 0,C 180,E1 -16951.275,E2 -16951.275} C_VEL
LIN {X 0,Y 284.358,Z 386.063,A -85,B 0,C 180,E1 -16955.355,E2 -16955.355} C_VEL
LIN {X 0,Y 284.333,Z 386.068,A -85,B 0,C 180,E1 -16958.165,E2 -16958.165} C_VEL
LIN {X 0,Y 284.339,Z 386.067,A -85,B 0,C 180,E1 -16962.141,E2 -16962.141} C_VEL
LIN {X 0,Y 284.294,Z 386.073,A -85,B 0,C 180,E1 -16966.198,E2 -16966.198} C_VEL
LIN {X 0,Y 284.331,Z 386.07,A -85,B 0,C 180,E1 -16970.018,E2 -16970.018} C_VEL
LIN {X 0,Y 284.348,Z 386.067,A -85,B 0,C 180,E1 -16973.617,E2 -16973.617} C_VEL
LIN {X 0,Y 284.387,Z 386.139,A -85,B 0,C 180,E1 -16976.06,E2 -16976.06} C_VEL
LIN {X 0,Y 286.881,Z 397.735,A -85,B 0,C 180,E1 -16979.855,E2 -16979.855} C_VEL
LIN {X 0,Y 288.682,Z 407.349,A -85,B 0,C 180,E1 -16982.841,E2 -16982.841} C_VEL
LIN {X 0,Y 288.548,Z 410.354,A -85,B 0,C 180,E1 -16983.707,E2 -16983.707} C_VEL
LIN {X 0,Y 293.226,Z 445.144,A -85,B 0,C 180,E1 -16984.996,E2 -16984.996} C_VEL
LIN {X 0,Y 294.699,Z 457.878,A -85,B 0,C 180,E1 -16985.434,E2 -16985.434} C_VEL
LIN {X 0,Y 293.121,Z 519.26,A -85,B 0,C 180,E1 -16986.93,E2 -16986.93} C_VEL
LIN {X 0,Y 292.378,Z 532.513,A -85,B 0,C 180,E1 -16987.522,E2 -16987.522} C_VEL
LIN {X 0,Y 291.307,Z 544.673,A -85,B 0,C 180,E1 -16988.32,E2 -16988.32} C_VEL
LIN {X 0,Y 289.952,Z 556.937,A -85,B 0,C 180,E1 -16989.424,E2 -16989.424} C_VEL
LIN {X 0,Y 288.394,Z 568.557,A -85,B 0,C 180,E1 -16990.793,E2 -16990.793} C_VEL
LIN {X 0,Y 286.949,Z 579.033,A -85,B 0,C 180,E1 -16992.357,E2 -16992.357} C_VEL
LIN {X 0,Y 285.868,Z 588.115,A -85,B 0,C 180,E1 -16994.052,E2 -16994.052} C_VEL
LIN {X 0,Y 284.612,Z 596.867,A -85,B 0,C 180,E1 -16996.069,E2 -16996.069} C_VEL
LIN {X 0,Y 283.537,Z 604.303,A -85,B 0,C 180,E1 -16998.201,E2 -16998.201} C_VEL
LIN {X 0,Y 283.044,Z 609.357,A -85,B 0,C 180,E1 -16999.991,E2 -16999.991} C_VEL
LIN {X 0,Y 282.635,Z 614.249,A -85,B 0,C 180,E1 -17002.14,E2 -17002.14} C_VEL
LIN {X 0,Y 282.463,Z 618.181,A -85,B 0,C 180,E1 -17004.41,E2 -17004.41} C_VEL
LIN {X 0,Y 282.437,Z 619.93,A -85,B 0,C 180,E1 -17005.719,E2 -17005.719} C_VEL
LIN {X 0,Y 282.463,Z 621.417,A -85,B 0,C 180,E1 -17007.148,E2 -17007.148} C_VEL
LIN {X 0,Y 282.464,Z 622.453,A -85,B 0,C 180,E1 -17008.574,E2 -17008.574} C_VEL
LIN {X 0,Y 282.496,Z 623.094,A -85,B 0,C 180,E1 -17010,E2 -17010} C_VEL
LIN {X 0,Y 282.43,Z 623.34,A -85,B 0,C 180,E1 -17011.426,E2 -17011.426} C_VEL
LIN {X 0,Y 282.43,Z 623.183,A -85,B 0,C 180,E1 -17012.853,E2 -17012.853} C_VEL
LIN {X 0,Y 282.384,Z 621.617,A -85,B 0,C 180,E1 -17015.713,E2 -17015.713} C_VEL
LIN {X 0,Y 282.506,Z 620.251,A -85,B 0,C 180,E1 -17017.145,E2 -17017.145} C_VEL
LIN {X 0,Y 282.954,Z 617.389,A -85,B 0,C 180,E1 -17019.291,E2 -17019.291} C_VEL
LIN {X 0,Y 283.65,Z 613.516,A -85,B 0,C 180,E1 -17021.432,E2 -17021.432} C_VEL
LIN {X 0,Y 284.717,Z 608.538,A -85,B 0,C 180,E1 -17023.562,E2 -17023.562} C_VEL
LIN {X 0,Y 286.252,Z 602.308,A -85,B 0,C 180,E1 -17025.668,E2 -17025.668} C_VEL
LIN {X 0,Y 287.856,Z 595.216,A -85,B 0,C 180,E1 -17027.603,E2 -17027.603} C_VEL
LIN {X 0,Y 289.703,Z 586.683,A -85,B 0,C 180,E1 -17029.485,E2 -17029.485} C_VEL
LIN {X 0,Y 291.891,Z 577.084,A -85,B 0,C 180,E1 -17031.171,E2 -17031.171} C_VEL
LIN {X 0,Y 294.089,Z 566.454,A -85,B 0,C 180,E1 -17032.665,E2 -17032.665} C_VEL
LIN {X 0,Y 295.962,Z 556.197,A -85,B 0,C 180,E1 -17033.808,E2 -17033.808} C_VEL
LIN {X 0,Y 297.673,Z 545.114,A -85,B 0,C 180,E1 -17034.775,E2 -17034.775} C_VEL
LIN {X 0,Y 299.18,Z 532.727,A -85,B 0,C 180,E1 -17035.571,E2 -17035.571} C_VEL
LIN {X 0,Y 300.315,Z 518.961,A -85,B 0,C 180,E1 -17036.166,E2 -17036.166} C_VEL
LIN {X 0,Y 302.237,Z 459.12,A -85,B 0,C 180,E1 -17037.619,E2 -17037.619} C_VEL
LIN {X 0,Y 298.597,Z 436.638,A -85,B 0,C 180,E1 -17038.66,E2 -17038.66} C_VEL
LIN {X 0,Y 295.371,Z 421.401,A -85,B 0,C 180,E1 -17039.481,E2 -17039.481} C_VEL
LIN {X 0,Y 289.958,Z 409.404,A -85,B 0,C 180,E1 -17040.537,E2 -17040.537} C_VEL
LIN {X 0,Y 287.683,Z 399.124,A -85,B 0,C 180,E1 -17044.185,E2 -17044.185} C_VEL
LIN {X 0,Y 285.552,Z 390.713,A -85,B 0,C 180,E1 -17047.389,E2 -17047.389} C_VEL
LIN {X 0,Y 284.33,Z 386.067,A -85,B 0,C 180,E1 -17049.3,E2 -17049.3} C_VEL
LIN {X 0,Y 284.294,Z 386.068,A -85,B 0,C 180,E1 -17053.802,E2 -17053.802} C_VEL
LIN {X 0,Y 284.336,Z 386.061,A -85,B 0,C 180,E1 -17058.136,E2 -17058.136} C_VEL
LIN {X 0,Y 284.342,Z 386.061,A -85,B 0,C 180,E1 -17062.271,E2 -17062.271} C_VEL
LIN {X 0,Y 284.319,Z 386.068,A -85,B 0,C 180,E1 -17065.352,E2 -17065.352} C_VEL
LIN {X 0,Y 284.291,Z 386.072,A -85,B 0,C 180,E1 -17068.725,E2 -17068.725} C_VEL
LIN {X 0,Y 284.392,Z 386.052,A -85,B 0,C 180,E1 -17072.826,E2 -17072.826} C_VEL
LIN {X 0,Y 284.36,Z 386.048,A -85,B 0,C 180,E1 -17076.707,E2 -17076.707} C_VEL
LIN {X 0,Y 284.397,Z 386.052,A -85,B 0,C 180,E1 -17081.261,E2 -17081.261} C_VEL
LIN {X 0,Y 284.472,Z 386.044,A -85,B 0,C 180,E1 -17084.47,E2 -17084.47} C_VEL
LIN {X 0,Y 284.484,Z 386.044,A -85,B 0,C 180,E1 -17088.602,E2 -17088.602} C_VEL
LIN {X 0,Y 284.653,Z 386.028,A -85,B 0,C 180,E1 -17091.481,E2 -17091.481} C_VEL
LIN {X 0,Y 284.596,Z 386.024,A -85,B 0,C 180,E1 -17094.331,E2 -17094.331} C_VEL
LIN {X 0,Y 284.851,Z 385.994,A -85,B 0,C 180,E1 -17098.587,E2 -17098.587} C_VEL
LIN {X 0,Y 284.851,Z 386.002,A -85,B 0,C 180,E1 -17101.414,E2 -17101.414} C_VEL
LIN {X 0,Y 284.681,Z 386.018,A -85,B 0,C 180,E1 -17107.091,E2 -17107.091} C_VEL
LIN {X 0,Y 284.513,Z 386.043,A -85,B 0,C 180,E1 -17109.958,E2 -17109.958} C_VEL
LIN {X 0,Y 284.472,Z 386.049,A -85,B 0,C 180,E1 -17114.304,E2 -17114.304} C_VEL
LIN {X 0,Y 284.42,Z 386.049,A -85,B 0,C 180,E1 -17117.249,E2 -17117.249} C_VEL
LIN {X 0,Y 284.374,Z 386.058,A -85,B 0,C 180,E1 -17120.243,E2 -17120.243} C_VEL
LIN {X 0,Y 284.364,Z 386.06,A -85,B 0,C 180,E1 -17123.876,E2 -17123.876} C_VEL
LIN {X 0,Y 284.391,Z 386.036,A -85,B 0,C 180,E1 -17127.174,E2 -17127.174} C_VEL
LIN {X 0,Y 284.292,Z 386.066,A -85,B 0,C 180,E1 -17131.275,E2 -17131.275} C_VEL
LIN {X 0,Y 284.36,Z 386.065,A -85,B 0,C 180,E1 -17135.355,E2 -17135.355} C_VEL
LIN {X 0,Y 284.334,Z 386.071,A -85,B 0,C 180,E1 -17138.166,E2 -17138.166} C_VEL
LIN {X 0,Y 284.339,Z 386.059,A -85,B 0,C 180,E1 -17142.141,E2 -17142.141} C_VEL
LIN {X 0,Y 284.317,Z 386.067,A -85,B 0,C 180,E1 -17146.203,E2 -17146.203} C_VEL
LIN {X 0,Y 284.351,Z 386.254,A -85,B 0,C 180,E1 -17149.125,E2 -17149.125} C_VEL
LIN {X 0,Y 284.871,Z 388.037,A -85,B 0,C 180,E1 -17149.836,E2 -17149.836} C_VEL
LIN {X 0,Y 295.019,Z 407.318,A -85,B 0,C 180,E1 -17151.762,E2 -17151.762} C_VEL
LIN {X 0,Y 301.898,Z 422.401,A -85,B 0,C 180,E1 -17153.027,E2 -17153.027} C_VEL
LIN {X 0,Y 303.352,Z 426.259,A -85,B 0,C 180,E1 -17153.303,E2 -17153.303} C_VEL
LIN {X 0,Y 301.052,Z 493.611,A -85,B 0,C 180,E1 -17154.91,E2 -17154.91} C_VEL
LIN {X 0,Y 300.21,Z 506.001,A -85,B 0,C 180,E1 -17155.439,E2 -17155.439} C_VEL
LIN {X 0,Y 298.951,Z 518.884,A -85,B 0,C 180,E1 -17156.263,E2 -17156.263} C_VEL
LIN {X 0,Y 297.246,Z 530.543,A -85,B 0,C 180,E1 -17157.259,E2 -17157.259} C_VEL
LIN {X 0,Y 295.673,Z 541.143,A -85,B 0,C 180,E1 -17158.472,E2 -17158.472} C_VEL
LIN {X 0,Y 293.679,Z 552,A -85,B 0,C 180,E1 -17160.03,E2 -17160.03} C_VEL
LIN {X 0,Y 291.752,Z 560.815,A -85,B 0,C 180,E1 -17161.592,E2 -17161.592} C_VEL
LIN {X 0,Y 289.853,Z 569.189,A -85,B 0,C 180,E1 -17163.427,E2 -17163.427} C_VEL
LIN {X 0,Y 288.008,Z 576.723,A -85,B 0,C 180,E1 -17165.492,E2 -17165.492} C_VEL
LIN {X 0,Y 286.334,Z 582.95,A -85,B 0,C 180,E1 -17167.639,E2 -17167.639} C_VEL
LIN {X 0,Y 285.033,Z 587.856,A -85,B 0,C 180,E1 -17169.807,E2 -17169.807} C_VEL
LIN {X 0,Y 284.054,Z 591.6,A -85,B 0,C 180,E1 -17171.985,E2 -17171.985} C_VEL
LIN {X 0,Y 283.357,Z 594.288,A -85,B 0,C 180,E1 -17174.168,E2 -17174.168} C_VEL
LIN {X 0,Y 283.028,Z 595.54,A -85,B 0,C 180,E1 -17175.623,E2 -17175.623} C_VEL
LIN {X 0,Y 282.725,Z 596.389,A -85,B 0,C 180,E1 -17177.073,E2 -17177.073} C_VEL
LIN {X 0,Y 282.384,Z 596.806,A -85,B 0,C 180,E1 -17179.967,E2 -17179.967} C_VEL
LIN {X 0,Y 282.394,Z 596.43,A -85,B 0,C 180,E1 -17181.412,E2 -17181.412} C_VEL
LIN {X 0,Y 282.605,Z 594.614,A -85,B 0,C 180,E1 -17184.13,E2 -17184.13} C_VEL
LIN {X 0,Y 282.77,Z 591.899,A -85,B 0,C 180,E1 -17186.438,E2 -17186.438} C_VEL
LIN {X 0,Y 283.218,Z 588.342,A -85,B 0,C 180,E1 -17188.578,E2 -17188.578} C_VEL
LIN {X 0,Y 283.691,Z 583.702,A -85,B 0,C 180,E1 -17190.71,E2 -17190.71} C_VEL
LIN {X 0,Y 284.704,Z 576.704,A -85,B 0,C 180,E1 -17193.184,E2 -17193.184} C_VEL
LIN {X 0,Y 285.878,Z 569.127,A -85,B 0,C 180,E1 -17195.289,E2 -17195.289} C_VEL
LIN {X 0,Y 287.23,Z 559.617,A -85,B 0,C 180,E1 -17197.38,E2 -17197.38} C_VEL
LIN {X 0,Y 288.652,Z 549.797,A -85,B 0,C 180,E1 -17199.106,E2 -17199.106} C_VEL
LIN {X 0,Y 290.082,Z 538.767,A -85,B 0,C 180,E1 -17200.645,E2 -17200.645} C_VEL
LIN {X 0,Y 291.391,Z 526.239,A -85,B 0,C 180,E1 -17202.006,E2 -17202.006} C_VEL
LIN {X 0,Y 292.376,Z 514.985,A -85,B 0,C 180,E1 -17202.935,E2 -17202.935} C_VEL
LIN {X 0,Y 293.183,Z 502.254,A -85,B 0,C 180,E1 -17203.693,E2 -17203.693} C_VEL
LIN {X 0,Y 293.695,Z 488.21,A -85,B 0,C 180,E1 -17204.217,E2 -17204.217} C_VEL
LIN {X 0,Y 295.529,Z 416.631,A -85,B 0,C 180,E1 -17205.923,E2 -17205.923} C_VEL
LIN {X 0,Y 288.866,Z 397.613,A -85,B 0,C 180,E1 -17206.956,E2 -17206.956} C_VEL
LIN {X 0,Y 284.553,Z 386.597,A -85,B 0,C 180,E1 -17207.658,E2 -17207.658} C_VEL
LIN {X 0,Y 284.439,Z 386.055,A -85,B 0,C 180,E1 -17207.99,E2 -17207.99} C_VEL
LIN {X 0,Y 284.332,Z 386.067,A -85,B 0,C 180,E1 -17211.762,E2 -17211.762} C_VEL
LIN {X 0,Y 284.352,Z 386.058,A -85,B 0,C 180,E1 -17214.845,E2 -17214.845} C_VEL
LIN {X 0,Y 284.372,Z 386.062,A -85,B 0,C 180,E1 -17218.005,E2 -17218.005} C_VEL
LIN {X 0,Y 284.299,Z 386.069,A -85,B 0,C 180,E1 -17221.273,E2 -17221.273} C_VEL
LIN {X 0,Y 284.342,Z 386.064,A -85,B 0,C 180,E1 -17225.347,E2 -17225.347} C_VEL
LIN {X 0,Y 284.319,Z 386.07,A -85,B 0,C 180,E1 -17228.167,E2 -17228.167} C_VEL
LIN {X 0,Y 284.283,Z 386.069,A -85,B 0,C 180,E1 -17232.126,E2 -17232.126} C_VEL
LIN {X 0,Y 284.317,Z 386.066,A -85,B 0,C 180,E1 -17236.2,E2 -17236.2} C_VEL
LIN {X 0,Y 284.35,Z 386.063,A -85,B 0,C 180,E1 -17240.012,E2 -17240.012} C_VEL
LIN {X 0,Y 284.353,Z 386.06,A -85,B 0,C 180,E1 -17243.616,E2 -17243.616} C_VEL
LIN {X 0,Y 284.304,Z 386.066,A -85,B 0,C 180,E1 -17247.189,E2 -17247.189} C_VEL
LIN {X 0,Y 284.334,Z 386.066,A -85,B 0,C 180,E1 -17250.597,E2 -17250.597} C_VEL
LIN {X 0,Y 284.372,Z 386.055,A -85,B 0,C 180,E1 -17253.585,E2 -17253.585} C_VEL
LIN {X 0,Y 284.361,Z 386.061,A -85,B 0,C 180,E1 -17256.753,E2 -17256.753} C_VEL
LIN {X 0,Y 283.635,Z 386.154,A -85,B 0,C 180,E1 -17257.936,E2 -17257.936} C_VEL
LIN {X 0,Y 280.781,Z 386.509,A -85,B 0,C 180,E1 -17259.864,E2 -17259.864} C_VEL
LIN {X 0,Y 278.412,Z 386.801,A -85,B 0,C 180,E1 -17261.429,E2 -17261.429} C_VEL
LIN {X 0,Y 277.422,Z 386.92,A -85,B 0,C 180,E1 -17262.642,E2 -17262.642} C_VEL
LIN {X 0,Y 277.352,Z 386.926,A -85,B 0,C 180,E1 -17263.052,E2 -17263.052} C_VEL
LIN {X 0,Y 277.412,Z 386.924,A -85,B 0,C 180,E1 -17266.82,E2 -17266.82} C_VEL
LIN {X 0,Y 277.61,Z 386.901,A -85,B 0,C 180,E1 -17271.263,E2 -17271.263} C_VEL
LIN {X 0,Y 277.566,Z 386.899,A -85,B 0,C 180,E1 -17274.187,E2 -17274.187} C_VEL
LIN {X 0,Y 277.816,Z 386.877,A -85,B 0,C 180,E1 -17278.55,E2 -17278.55} C_VEL
LIN {X 0,Y 277.816,Z 386.877,A -85,B 0,C 180,E1 -17281.449,E2 -17281.449} C_VEL
LIN {X 0,Y 277.647,Z 386.897,A -85,B 0,C 180,E1 -17287.271,E2 -17287.271} C_VEL
LIN {X 0,Y 277.501,Z 386.92,A -85,B 0,C 180,E1 -17290.211,E2 -17290.211} C_VEL
LIN {X 0,Y 277.423,Z 386.926,A -85,B 0,C 180,E1 -17294.674,E2 -17294.674} C_VEL
LIN {X 0,Y 277.341,Z 386.934,A -85,B 0,C 180,E1 -17299.234,E2 -17299.234} C_VEL
LIN {X 0,Y 277.323,Z 386.94,A -85,B 0,C 180,E1 -17303.921,E2 -17303.921} C_VEL
LIN {X 0,Y 277.318,Z 386.94,A -85,B 0,C 180,E1 -17307.504,E2 -17307.504} C_VEL
LIN {X 0,Y 277.267,Z 386.947,A -85,B 0,C 180,E1 -17310.482,E2 -17310.482} C_VEL
LIN {X 0,Y 277.249,Z 386.952,A -85,B 0,C 180,E1 -17313.895,E2 -17313.895} C_VEL
LIN {X 0,Y 277.286,Z 386.945,A -85,B 0,C 180,E1 -17317.466,E2 -17317.466} C_VEL
LIN {X 0,Y 277.262,Z 386.947,A -85,B 0,C 180,E1 -17321.227,E2 -17321.227} C_VEL
LIN {X 0,Y 277.24,Z 386.948,A -85,B 0,C 180,E1 -17325.218,E2 -17325.218} C_VEL
LIN {X 0,Y 277.247,Z 386.951,A -85,B 0,C 180,E1 -17329.506,E2 -17329.506} C_VEL
LIN {X 0,Y 277.279,Z 386.945,A -85,B 0,C 180,E1 -17332.533,E2 -17332.533} C_VEL
LIN {X 0,Y 277.328,Z 387.109,A -85,B 0,C 180,E1 -17335.623,E2 -17335.623} C_VEL
LIN {X 0,Y 279.736,Z 398.106,A -85,B 0,C 180,E1 -17339.339,E2 -17339.339} C_VEL
LIN {X 0,Y 281.652,Z 407.979,A -85,B 0,C 180,E1 -17342.509,E2 -17342.509} C_VEL
LIN {X 0,Y 281.767,Z 410.004,A -85,B 0,C 180,E1 -17343.123,E2 -17343.123} C_VEL
LIN {X 0,Y 286.503,Z 444.706,A -85,B 0,C 180,E1 -17344.461,E2 -17344.461} C_VEL
LIN {X 0,Y 288.043,Z 458.757,A -85,B 0,C 180,E1 -17344.954,E2 -17344.954} C_VEL
LIN {X 0,Y 286.444,Z 519.161,A -85,B 0,C 180,E1 -17346.462,E2 -17346.462} C_VEL
LIN {X 0,Y 285.673,Z 532.229,A -85,B 0,C 180,E1 -17347.06,E2 -17347.06} C_VEL
LIN {X 0,Y 284.549,Z 544.372,A -85,B 0,C 180,E1 -17347.874,E2 -17347.874} C_VEL
LIN {X 0,Y 283.27,Z 555.825,A -85,B 0,C 180,E1 -17348.916,E2 -17348.916} C_VEL
LIN {X 0,Y 281.703,Z 567.6,A -85,B 0,C 180,E1 -17350.318,E2 -17350.318} C_VEL
LIN {X 0,Y 280.268,Z 577.091,A -85,B 0,C 180,E1 -17351.733,E2 -17351.733} C_VEL
LIN {X 0,Y 278.997,Z 587.09,A -85,B 0,C 180,E1 -17353.59,E2 -17353.59} C_VEL
LIN {X 0,Y 277.665,Z 596.201,A -85,B 0,C 180,E1 -17355.713,E2 -17355.713} C_VEL
LIN {X 0,Y 276.559,Z 603.697,A -85,B 0,C 180,E1 -17357.898,E2 -17357.898} C_VEL
LIN {X 0,Y 275.842,Z 610.605,A -85,B 0,C 180,E1 -17360.468,E2 -17360.468} C_VEL
LIN {X 0,Y 275.493,Z 615.146,A -85,B 0,C 180,E1 -17362.672,E2 -17362.672} C_VEL
LIN {X 0,Y 275.374,Z 618.018,A -85,B 0,C 180,E1 -17364.469,E2 -17364.469} C_VEL
LIN {X 0,Y 275.389,Z 621.013,A -85,B 0,C 180,E1 -17367.074,E2 -17367.074} C_VEL
LIN {X 0,Y 275.383,Z 622.072,A -85,B 0,C 180,E1 -17368.538,E2 -17368.538} C_VEL
LIN {X 0,Y 275.411,Z 622.732,A -85,B 0,C 180,E1 -17370,E2 -17370} C_VEL
LIN {X 0,Y 275.351,Z 622.996,A -85,B 0,C 180,E1 -17371.463,E2 -17371.463} C_VEL
LIN {X 0,Y 275.355,Z 622.87,A -85,B 0,C 180,E1 -17372.926,E2 -17372.926} C_VEL
LIN {X 0,Y 275.331,Z 621.684,A -85,B 0,C 180,E1 -17375.438,E2 -17375.438} C_VEL
LIN {X 0,Y 275.455,Z 620.003,A -85,B 0,C 180,E1 -17377.329,E2 -17377.329} C_VEL
LIN {X 0,Y 275.922,Z 617.181,A -85,B 0,C 180,E1 -17379.53,E2 -17379.53} C_VEL
LIN {X 0,Y 276.641,Z 613.351,A -85,B 0,C 180,E1 -17381.726,E2 -17381.726} C_VEL
LIN {X 0,Y 277.809,Z 608.42,A -85,B 0,C 180,E1 -17383.906,E2 -17383.906} C_VEL
LIN {X 0,Y 279.386,Z 602.241,A -85,B 0,C 180,E1 -17386.063,E2 -17386.063} C_VEL
LIN {X 0,Y 281.294,Z 594.178,A -85,B 0,C 180,E1 -17388.302,E2 -17388.302} C_VEL
LIN {X 0,Y 283.43,Z 584.995,A -85,B 0,C 180,E1 -17390.312,E2 -17390.312} C_VEL
LIN {X 0,Y 285.792,Z 575.127,A -85,B 0,C 180,E1 -17392.025,E2 -17392.025} C_VEL
LIN {X 0,Y 288.04,Z 564.083,A -85,B 0,C 180,E1 -17393.549,E2 -17393.549} C_VEL
LIN {X 0,Y 290.013,Z 553.286,A -85,B 0,C 180,E1 -17394.709,E2 -17394.709} C_VEL
LIN {X 0,Y 292.016,Z 540.273,A -85,B 0,C 180,E1 -17395.766,E2 -17395.766} C_VEL
LIN {X 0,Y 293.47,Z 527.648,A -85,B 0,C 180,E1 -17396.489,E2 -17396.489} C_VEL
LIN {X 0,Y 294.414,Z 514.446,A -85,B 0,C 180,E1 -17396.971,E2 -17396.971} C_VEL
LIN {X 0,Y 296.136,Z 460.103,A -85,B 0,C 180,E1 -17398.298,E2 -17398.298} C_VEL
LIN {X 0,Y 292.497,Z 437.498,A -85,B 0,C 180,E1 -17399.382,E2 -17399.382} C_VEL
LIN {X 0,Y 289.731,Z 424.43,A -85,B 0,C 180,E1 -17400.112,E2 -17400.112} C_VEL
LIN {X 0,Y 284.092,Z 412.341,A -85,B 0,C 180,E1 -17401.228,E2 -17401.228} C_VEL
LIN {X 0,Y 282.656,Z 408.878,A -85,B 0,C 180,E1 -17401.58,E2 -17401.58} C_VEL
LIN {X 0,Y 280.808,Z 400.648,A -85,B 0,C 180,E1 -17404.618,E2 -17404.618} C_VEL
LIN {X 0,Y 278.626,Z 392.064,A -85,B 0,C 180,E1 -17408.003,E2 -17408.003} C_VEL
LIN {X 0,Y 277.242,Z 386.949,A -85,B 0,C 180,E1 -17410.194,E2 -17410.194} C_VEL
LIN {X 0,Y 277.233,Z 386.946,A -85,B 0,C 180,E1 -17413.192,E2 -17413.192} C_VEL
LIN {X 0,Y 277.268,Z 386.941,A -85,B 0,C 180,E1 -17417.312,E2 -17417.312} C_VEL
LIN {X 0,Y 277.264,Z 386.943,A -85,B 0,C 180,E1 -17420.677,E2 -17420.677} C_VEL
LIN {X 0,Y 277.301,Z 386.94,A -85,B 0,C 180,E1 -17424.344,E2 -17424.344} C_VEL
LIN {X 0,Y 277.24,Z 386.952,A -85,B 0,C 180,E1 -17427.836,E2 -17427.836} C_VEL
LIN {X 0,Y 277.284,Z 386.945,A -85,B 0,C 180,E1 -17431.212,E2 -17431.212} C_VEL
LIN {X 0,Y 277.308,Z 386.913,A -85,B 0,C 180,E1 -17434.479,E2 -17434.479} C_VEL
LIN {X 0,Y 277.28,Z 386.94,A -85,B 0,C 180,E1 -17437.655,E2 -17437.655} C_VEL
LIN {X 0,Y 277.339,Z 386.93,A -85,B 0,C 180,E1 -17440.766,E2 -17440.766} C_VEL
LIN {X 0,Y 277.423,Z 386.92,A -85,B 0,C 180,E1 -17445.326,E2 -17445.326} C_VEL
LIN {X 0,Y 277.501,Z 386.909,A -85,B 0,C 180,E1 -17449.789,E2 -17449.789} C_VEL
LIN {X 0,Y 277.646,Z 386.898,A -85,B 0,C 180,E1 -17452.729,E2 -17452.729} C_VEL
LIN {X 0,Y 277.816,Z 386.87,A -85,B 0,C 180,E1 -17458.551,E2 -17458.551} C_VEL
LIN {X 0,Y 277.816,Z 386.878,A -85,B 0,C 180,E1 -17461.45,E2 -17461.45} C_VEL
LIN {X 0,Y 277.635,Z 386.895,A -85,B 0,C 180,E1 -17467.272,E2 -17467.272} C_VEL
LIN {X 0,Y 277.455,Z 386.924,A -85,B 0,C 180,E1 -17470.214,E2 -17470.214} C_VEL
LIN {X 0,Y 277.423,Z 386.93,A -85,B 0,C 180,E1 -17474.675,E2 -17474.675} C_VEL
LIN {X 0,Y 277.341,Z 386.938,A -85,B 0,C 180,E1 -17479.235,E2 -17479.235} C_VEL
LIN {X 0,Y 277.314,Z 386.934,A -85,B 0,C 180,E1 -17484.171,E2 -17484.171} C_VEL
LIN {X 0,Y 277.32,Z 386.919,A -85,B 0,C 180,E1 -17487.505,E2 -17487.505} C_VEL
LIN {X 0,Y 277.269,Z 386.944,A -85,B 0,C 180,E1 -17490.482,E2 -17490.482} C_VEL
LIN {X 0,Y 277.252,Z 386.947,A -85,B 0,C 180,E1 -17493.896,E2 -17493.896} C_VEL
LIN {X 0,Y 277.288,Z 386.945,A -85,B 0,C 180,E1 -17497.467,E2 -17497.467} C_VEL
LIN {X 0,Y 277.291,Z 386.945,A -85,B 0,C 180,E1 -17501.223,E2 -17501.223} C_VEL
LIN {X 0,Y 277.25,Z 386.953,A -85,B 0,C 180,E1 -17505.217,E2 -17505.217} C_VEL
LIN {X 0,Y 277.31,Z 387.13,A -85,B 0,C 180,E1 -17508.284,E2 -17508.284} C_VEL
LIN {X 0,Y 277.629,Z 388.354,A -85,B 0,C 180,E1 -17508.786,E2 -17508.786} C_VEL
LIN {X 0,Y 286.581,Z 404.83,A -85,B 0,C 180,E1 -17510.579,E2 -17510.579} C_VEL
LIN {X 0,Y 294.183,Z 420.521,A -85,B 0,C 180,E1 -17512.034,E2 -17512.034} C_VEL
LIN {X 0,Y 297.214,Z 427.735,A -85,B 0,C 180,E1 -17512.614,E2 -17512.614} C_VEL
LIN {X 0,Y 294.936,Z 493.761,A -85,B 0,C 180,E1 -17514.224,E2 -17514.224} C_VEL
LIN {X 0,Y 294.067,Z 506.198,A -85,B 0,C 180,E1 -17514.761,E2 -17514.761} C_VEL
LIN {X 0,Y 292.674,Z 519.759,A -85,B 0,C 180,E1 -17515.647,E2 -17515.647} C_VEL
LIN {X 0,Y 290.906,Z 531.264,A -85,B 0,C 180,E1 -17516.66,E2 -17516.66} C_VEL
LIN {X 0,Y 289.173,Z 542.35,A -85,B 0,C 180,E1 -17517.973,E2 -17517.973} C_VEL
LIN {X 0,Y 287.182,Z 552.581,A -85,B 0,C 180,E1 -17519.483,E2 -17519.483} C_VEL
LIN {X 0,Y 284.981,Z 562.252,A -85,B 0,C 180,E1 -17521.257,E2 -17521.257} C_VEL
LIN {X 0,Y 283.077,Z 570.113,A -85,B 0,C 180,E1 -17523.058,E2 -17523.058} C_VEL
LIN {X 0,Y 281.099,Z 577.747,A -85,B 0,C 180,E1 -17525.243,E2 -17525.243} C_VEL
LIN {X 0,Y 279.112,Z 584.75,A -85,B 0,C 180,E1 -17527.809,E2 -17527.809} C_VEL
LIN {X 0,Y 277.853,Z 589.332,A -85,B 0,C 180,E1 -17530.034,E2 -17530.034} C_VEL
LIN {X 0,Y 276.87,Z 592.783,A -85,B 0,C 180,E1 -17532.266,E2 -17532.266} C_VEL
LIN {X 0,Y 276.392,Z 594.483,A -85,B 0,C 180,E1 -17533.758,E2 -17533.758} C_VEL
LIN {X 0,Y 276,Z 595.867,A -85,B 0,C 180,E1 -17535.383,E2 -17535.383} C_VEL
LIN {X 0,Y 275.458,Z 597.115,A -85,B 0,C 180,E1 -17538.223,E2 -17538.223} C_VEL
LIN {X 0,Y 275.302,Z 596.813,A -85,B 0,C 180,E1 -17541.19,E2 -17541.19} C_VEL
LIN {X 0,Y 275.358,Z 596.085,A -85,B 0,C 180,E1 -17542.668,E2 -17542.668} C_VEL
LIN {X 0,Y 275.533,Z 594.925,A -85,B 0,C 180,E1 -17544.144,E2 -17544.144} C_VEL
LIN {X 0,Y 275.605,Z 593.355,A -85,B 0,C 180,E1 -17545.613,E2 -17545.613} C_VEL
LIN {X 0,Y 275.923,Z 590.206,A -85,B 0,C 180,E1 -17547.81,E2 -17547.81} C_VEL
LIN {X 0,Y 276.411,Z 586.01,A -85,B 0,C 180,E1 -17550,E2 -17550} C_VEL
LIN {X 0,Y 277.309,Z 579.64,A -85,B 0,C 180,E1 -17552.542,E2 -17552.542} C_VEL
LIN {X 0,Y 278.408,Z 572.684,A -85,B 0,C 180,E1 -17554.706,E2 -17554.706} C_VEL
LIN {X 0,Y 279.753,Z 563.981,A -85,B 0,C 180,E1 -17556.853,E2 -17556.853} C_VEL
LIN {X 0,Y 281.066,Z 555.079,A -85,B 0,C 180,E1 -17558.628,E2 -17558.628} C_VEL
LIN {X 0,Y 282.525,Z 545.273,A -85,B 0,C 180,E1 -17560.209,E2 -17560.209} C_VEL
LIN {X 0,Y 283.84,Z 534.454,A -85,B 0,C 180,E1 -17561.606,E2 -17561.606} C_VEL
LIN {X 0,Y 284.989,Z 522.37,A -85,B 0,C 180,E1 -17562.823,E2 -17562.823} C_VEL
LIN {X 0,Y 286.12,Z 509.644,A -85,B 0,C 180,E1 -17563.766,E2 -17563.766} C_VEL
LIN {X 0,Y 286.787,Z 496.385,A -85,B 0,C 180,E1 -17564.435,E2 -17564.435} C_VEL
LIN {X 0,Y 287.298,Z 478.312,A -85,B 0,C 180,E1 -17564.949,E2 -17564.949} C_VEL
LIN {X 0,Y 288.819,Z 417.692,A -85,B 0,C 180,E1 -17566.428,E2 -17566.428} C_VEL
LIN {X 0,Y 281.93,Z 398.325,A -85,B 0,C 180,E1 -17567.529,E2 -17567.529} C_VEL
LIN {X 0,Y 277.482,Z 387.487,A -85,B 0,C 180,E1 -17568.227,E2 -17568.227} C_VEL
LIN {X 0,Y 277.392,Z 386.934,A -85,B 0,C 180,E1 -17568.32,E2 -17568.32} C_VEL
LIN {X 0,Y 277.289,Z 386.946,A -85,B 0,C 180,E1 -17572.344,E2 -17572.344} C_VEL
LIN {X 0,Y 277.322,Z 386.932,A -85,B 0,C 180,E1 -17575.519,E2 -17575.519} C_VEL
LIN {X 0,Y 277.31,Z 386.941,A -85,B 0,C 180,E1 -17578.784,E2 -17578.784} C_VEL
LIN {X 0,Y 277.255,Z 386.947,A -85,B 0,C 180,E1 -17583.226,E2 -17583.226} C_VEL
LIN {X 0,Y 277.282,Z 386.944,A -85,B 0,C 180,E1 -17585.798,E2 -17585.798} C_VEL
LIN {X 0,Y 277.237,Z 386.948,A -85,B 0,C 180,E1 -17589.327,E2 -17589.327} C_VEL
LIN {X 0,Y 277.235,Z 386.948,A -85,B 0,C 180,E1 -17593.192,E2 -17593.192} C_VEL
LIN {X 0,Y 277.271,Z 386.936,A -85,B 0,C 180,E1 -17597.311,E2 -17597.311} C_VEL
LIN {X 0,Y 277.267,Z 386.947,A -85,B 0,C 180,E1 -17600.677,E2 -17600.677} C_VEL
LIN {X 0,Y 277.303,Z 386.935,A -85,B 0,C 180,E1 -17604.344,E2 -17604.344} C_VEL
LIN {X 0,Y 277.24,Z 386.947,A -85,B 0,C 180,E1 -17607.835,E2 -17607.835} C_VEL
LIN {X 0,Y 277.264,Z 386.944,A -85,B 0,C 180,E1 -17611.209,E2 -17611.209} C_VEL
LIN {X 0,Y 277.308,Z 386.933,A -85,B 0,C 180,E1 -17614.478,E2 -17614.478} C_VEL
LIN {X 0,Y 277.288,Z 386.941,A -85,B 0,C 180,E1 -17617.655,E2 -17617.655} C_VEL
LIN {X 0,Y 277.342,Z 386.935,A -85,B 0,C 180,E1 -17620.765,E2 -17620.765} C_VEL
LIN {X 0,Y 277.352,Z 386.926,A -85,B 0,C 180,E1 -17623.052,E2 -17623.052} C_VEL
LIN {X 0,Y 276.706,Z 387.008,A -85,B 0,C 180,E1 -17624.264,E2 -17624.264} C_VEL
LIN {X 0,Y 273.851,Z 387.366,A -85,B 0,C 180,E1 -17626.239,E2 -17626.239} C_VEL
LIN {X 0,Y 271.454,Z 387.668,A -85,B 0,C 180,E1 -17627.843,E2 -17627.843} C_VEL
LIN {X 0,Y 270.483,Z 387.79,A -85,B 0,C 180,E1 -17629.087,E2 -17629.087} C_VEL
LIN {X 0,Y 270.436,Z 387.796,A -85,B 0,C 180,E1 -17629.508,E2 -17629.508} C_VEL
LIN {X 0,Y 270.605,Z 387.77,A -85,B 0,C 180,E1 -17632.538,E2 -17632.538} C_VEL
LIN {X 0,Y 270.782,Z 387.753,A -85,B 0,C 180,E1 -17638.512,E2 -17638.512} C_VEL
LIN {X 0,Y 270.782,Z 387.753,A -85,B 0,C 180,E1 -17641.487,E2 -17641.487} C_VEL
LIN {X 0,Y 270.605,Z 387.775,A -85,B 0,C 180,E1 -17647.461,E2 -17647.461} C_VEL
LIN {X 0,Y 270.436,Z 387.798,A -85,B 0,C 180,E1 -17650.481,E2 -17650.481} C_VEL
LIN {X 0,Y 270.391,Z 387.801,A -85,B 0,C 180,E1 -17655.065,E2 -17655.065} C_VEL
LIN {X 0,Y 270.297,Z 387.813,A -85,B 0,C 180,E1 -17659.756,E2 -17659.756} C_VEL
LIN {X 0,Y 270.269,Z 387.818,A -85,B 0,C 180,E1 -17664.586,E2 -17664.586} C_VEL
LIN {X 0,Y 270.265,Z 387.82,A -85,B 0,C 180,E1 -17667.909,E2 -17667.909} C_VEL
LIN {X 0,Y 270.179,Z 387.83,A -85,B 0,C 180,E1 -17671.349,E2 -17671.349} C_VEL
LIN {X 0,Y 270.211,Z 387.825,A -85,B 0,C 180,E1 -17674.904,E2 -17674.904} C_VEL
LIN {X 0,Y 270.218,Z 387.824,A -85,B 0,C 180,E1 -17678.718,E2 -17678.718} C_VEL
LIN {X 0,Y 270.22,Z 387.824,A -85,B 0,C 180,E1 -17682.549,E2 -17682.549} C_VEL
LIN {X 0,Y 270.19,Z 387.828,A -85,B 0,C 180,E1 -17686.745,E2 -17686.745} C_VEL
LIN {X 0,Y 270.199,Z 387.829,A -85,B 0,C 180,E1 -17689.44,E2 -17689.44} C_VEL
LIN {X 0,Y 270.253,Z 387.823,A -85,B 0,C 180,E1 -17693.723,E2 -17693.723} C_VEL
LIN {X 0,Y 270.256,Z 387.89,A -85,B 0,C 180,E1 -17695.104,E2 -17695.104} C_VEL
LIN {X 0,Y 272.693,Z 399.007,A -85,B 0,C 180,E1 -17698.973,E2 -17698.973} C_VEL
LIN {X 0,Y 274.767,Z 409.744,A -85,B 0,C 180,E1 -17702.507,E2 -17702.507} C_VEL
LIN {X 0,Y 276.571,Z 419.751,A -85,B 0,C 180,E1 -17702.949,E2 -17702.949} C_VEL
LIN {X 0,Y 281.325,Z 457.61,A -85,B 0,C 180,E1 -17704.39,E2 -17704.39} C_VEL
LIN {X 0,Y 280.072,Z 511.782,A -85,B 0,C 180,E1 -17705.751,E2 -17705.751} C_VEL
LIN {X 0,Y 279.526,Z 525.298,A -85,B 0,C 180,E1 -17706.235,E2 -17706.235} C_VEL
LIN {X 0,Y 278.439,Z 538.188,A -85,B 0,C 180,E1 -17706.969,E2 -17706.969} C_VEL
LIN {X 0,Y 277.287,Z 549.202,A -85,B 0,C 180,E1 -17707.852,E2 -17707.852} C_VEL
LIN {X 0,Y 275.734,Z 561.025,A -85,B 0,C 180,E1 -17709.094,E2 -17709.094} C_VEL
LIN {X 0,Y 274.158,Z 571.663,A -85,B 0,C 180,E1 -17710.534,E2 -17710.534} C_VEL
LIN {X 0,Y 272.58,Z 582.438,A -85,B 0,C 180,E1 -17712.375,E2 -17712.375} C_VEL
LIN {X 0,Y 271.438,Z 591.098,A -85,B 0,C 180,E1 -17714.225,E2 -17714.225} C_VEL
LIN {X 0,Y 270.13,Z 599.518,A -85,B 0,C 180,E1 -17716.459,E2 -17716.459} C_VEL
LIN {X 0,Y 269.188,Z 606.298,A -85,B 0,C 180,E1 -17718.708,E2 -17718.708} C_VEL
LIN {X 0,Y 268.646,Z 611.711,A -85,B 0,C 180,E1 -17720.969,E2 -17720.969} C_VEL
LIN {X 0,Y 268.327,Z 615.918,A -85,B 0,C 180,E1 -17723.231,E2 -17723.231} C_VEL
LIN {X 0,Y 268.252,Z 619.046,A -85,B 0,C 180,E1 -17725.492,E2 -17725.492} C_VEL
LIN {X 0,Y 268.316,Z 620.6,A -85,B 0,C 180,E1 -17726.997,E2 -17726.997} C_VEL
LIN {X 0,Y 268.305,Z 621.69,A -85,B 0,C 180,E1 -17728.499,E2 -17728.499} C_VEL
LIN {X 0,Y 268.328,Z 622.37,A -85,B 0,C 180,E1 -17730,E2 -17730} C_VEL
LIN {X 0,Y 268.273,Z 622.653,A -85,B 0,C 180,E1 -17731.501,E2 -17731.501} C_VEL
LIN {X 0,Y 268.259,Z 622.549,A -85,B 0,C 180,E1 -17733.003,E2 -17733.003} C_VEL
LIN {X 0,Y 268.232,Z 621.553,A -85,B 0,C 180,E1 -17735.349,E2 -17735.349} C_VEL
LIN {X 0,Y 268.38,Z 619.755,A -85,B 0,C 180,E1 -17737.523,E2 -17737.523} C_VEL
LIN {X 0,Y 268.891,Z 616.974,A -85,B 0,C 180,E1 -17739.781,E2 -17739.781} C_VEL
LIN {X 0,Y 269.642,Z 613.186,A -85,B 0,C 180,E1 -17742.035,E2 -17742.035} C_VEL
LIN {X 0,Y 270.915,Z 608.303,A -85,B 0,C 180,E1 -17744.267,E2 -17744.267} C_VEL
LIN {X 0,Y 272.528,Z 602.176,A -85,B 0,C 180,E1 -17746.479,E2 -17746.479} C_VEL
LIN {X 0,Y 274.399,Z 594.77,A -85,B 0,C 180,E1 -17748.62,E2 -17748.62} C_VEL
LIN {X 0,Y 276.347,Z 586.861,A -85,B 0,C 180,E1 -17750.468,E2 -17750.468} C_VEL
LIN {X 0,Y 278.97,Z 576.391,A -85,B 0,C 180,E1 -17752.398,E2 -17752.398} C_VEL
LIN {X 0,Y 281.299,Z 565.763,A -85,B 0,C 180,E1 -17753.953,E2 -17753.953} C_VEL
LIN {X 0,Y 283.364,Z 555.503,A -85,B 0,C 180,E1 -17755.133,E2 -17755.133} C_VEL
LIN {X 0,Y 285.249,Z 544.413,A -85,B 0,C 180,E1 -17756.129,E2 -17756.129} C_VEL
LIN {X 0,Y 286.837,Z 532.025,A -85,B 0,C 180,E1 -17756.954,E2 -17756.954} C_VEL
LIN {X 0,Y 288.053,Z 518.252,A -85,B 0,C 180,E1 -17757.568,E2 -17757.568} C_VEL
LIN {X 0,Y 290.108,Z 461.099,A -85,B 0,C 180,E1 -17759.002,E2 -17759.002} C_VEL
LIN {X 0,Y 286.133,Z 436.56,A -85,B 0,C 180,E1 -17760.228,E2 -17760.228} C_VEL
LIN {X 0,Y 284.17,Z 427.542,A -85,B 0,C 180,E1 -17760.76,E2 -17760.76} C_VEL
LIN {X 0,Y 278.705,Z 415.712,A -85,B 0,C 180,E1 -17761.889,E2 -17761.889} C_VEL
LIN {X 0,Y 275.387,Z 408.552,A -85,B 0,C 180,E1 -17762.63,E2 -17762.63} C_VEL
LIN {X 0,Y 273.242,Z 399.135,A -85,B 0,C 180,E1 -17766.268,E2 -17766.268} C_VEL
LIN {X 0,Y 270.951,Z 390.481,A -85,B 0,C 180,E1 -17769.904,E2 -17769.904} C_VEL
LIN {X 0,Y 270.183,Z 387.826,A -85,B 0,C 180,E1 -17771.108,E2 -17771.108} C_VEL
LIN {X 0,Y 270.191,Z 387.823,A -85,B 0,C 180,E1 -17775.388,E2 -17775.388} C_VEL
LIN {X 0,Y 270.243,Z 387.818,A -85,B 0,C 180,E1 -17779.447,E2 -17779.447} C_VEL
LIN {X 0,Y 270.253,Z 387.819,A -85,B 0,C 180,E1 -17783.721,E2 -17783.721} C_VEL
LIN {X 0,Y 270.2,Z 387.827,A -85,B 0,C 180,E1 -17786.892,E2 -17786.892} C_VEL
LIN {X 0,Y 270.224,Z 387.821,A -85,B 0,C 180,E1 -17790.386,E2 -17790.386} C_VEL
LIN {X 0,Y 270.258,Z 387.798,A -85,B 0,C 180,E1 -17793.764,E2 -17793.764} C_VEL
LIN {X 0,Y 270.227,Z 387.812,A -85,B 0,C 180,E1 -17797.039,E2 -17797.039} C_VEL
LIN {X 0,Y 270.296,Z 387.809,A -85,B 0,C 180,E1 -17800.244,E2 -17800.244} C_VEL
LIN {X 0,Y 270.391,Z 387.795,A -85,B 0,C 180,E1 -17804.935,E2 -17804.935} C_VEL
LIN {X 0,Y 270.436,Z 387.789,A -85,B 0,C 180,E1 -17809.519,E2 -17809.519} C_VEL
LIN {X 0,Y 270.605,Z 387.777,A -85,B 0,C 180,E1 -17812.539,E2 -17812.539} C_VEL
LIN {X 0,Y 270.782,Z 387.746,A -85,B 0,C 180,E1 -17818.513,E2 -17818.513} C_VEL
LIN {X 0,Y 270.782,Z 387.754,A -85,B 0,C 180,E1 -17821.488,E2 -17821.488} C_VEL
LIN {X 0,Y 270.593,Z 387.771,A -85,B 0,C 180,E1 -17827.462,E2 -17827.462} C_VEL
LIN {X 0,Y 270.407,Z 387.803,A -85,B 0,C 180,E1 -17830.483,E2 -17830.483} C_VEL
LIN {X 0,Y 270.391,Z 387.804,A -85,B 0,C 180,E1 -17835.066,E2 -17835.066} C_VEL
LIN {X 0,Y 270.297,Z 387.815,A -85,B 0,C 180,E1 -17839.756,E2 -17839.756} C_VEL
LIN {X 0,Y 270.27,Z 387.807,A -85,B 0,C 180,E1 -17844.587,E2 -17844.587} C_VEL
LIN {X 0,Y 270.268,Z 387.802,A -85,B 0,C 180,E1 -17847.91,E2 -17847.91} C_VEL
LIN {X 0,Y 270.181,Z 387.824,A -85,B 0,C 180,E1 -17851.349,E2 -17851.349} C_VEL
LIN {X 0,Y 270.213,Z 387.826,A -85,B 0,C 180,E1 -17854.904,E2 -17854.904} C_VEL
LIN {X 0,Y 270.221,Z 387.826,A -85,B 0,C 180,E1 -17858.718,E2 -17858.718} C_VEL
LIN {X 0,Y 270.247,Z 387.814,A -85,B 0,C 180,E1 -17862.545,E2 -17862.545} C_VEL
LIN {X 0,Y 270.235,Z 387.887,A -85,B 0,C 180,E1 -17867.324,E2 -17867.324} C_VEL
LIN {X 0,Y 270.362,Z 388.59,A -85,B 0,C 180,E1 -17867.656,E2 -17867.656} C_VEL
LIN {X 0,Y 271.63,Z 391.259,A -85,B 0,C 180,E1 -17867.948,E2 -17867.948} C_VEL
LIN {X 0,Y 273.525,Z 394.236,A -85,B 0,C 180,E1 -17868.343,E2 -17868.343} C_VEL
LIN {X 0,Y 281.082,Z 407.959,A -85,B 0,C 180,E1 -17869.903,E2 -17869.903} C_VEL
LIN {X 0,Y 288.682,Z 423.828,A -85,B 0,C 180,E1 -17871.423,E2 -17871.423} C_VEL
LIN {X 0,Y 291.174,Z 429.726,A -85,B 0,C 180,E1 -17871.917,E2 -17871.917} C_VEL
LIN {X 0,Y 288.776,Z 495.055,A -85,B 0,C 180,E1 -17873.548,E2 -17873.548} C_VEL
LIN {X 0,Y 287.829,Z 507.715,A -85,B 0,C 180,E1 -17874.126,E2 -17874.126} C_VEL
LIN {X 0,Y 286.42,Z 520.634,A -85,B 0,C 180,E1 -17875.002,E2 -17875.002} C_VEL
LIN {X 0,Y 284.586,Z 531.979,A -85,B 0,C 180,E1 -17876.032,E2 -17876.032} C_VEL
LIN {X 0,Y 282.756,Z 543.083,A -85,B 0,C 180,E1 -17877.382,E2 -17877.382} C_VEL
LIN {X 0,Y 280.701,Z 553.172,A -85,B 0,C 180,E1 -17878.91,E2 -17878.91} C_VEL
LIN {X 0,Y 278.606,Z 561.9,A -85,B 0,C 180,E1 -17880.535,E2 -17880.535} C_VEL
LIN {X 0,Y 276.606,Z 569.901,A -85,B 0,C 180,E1 -17882.375,E2 -17882.375} C_VEL
LIN {X 0,Y 274.504,Z 577.649,A -85,B 0,C 180,E1 -17884.606,E2 -17884.606} C_VEL
LIN {X 0,Y 272.941,Z 582.913,A -85,B 0,C 180,E1 -17886.478,E2 -17886.478} C_VEL
LIN {X 0,Y 271.41,Z 588.037,A -85,B 0,C 180,E1 -17888.782,E2 -17888.782} C_VEL
LIN {X 0,Y 270.271,Z 591.856,A -85,B 0,C 180,E1 -17891.032,E2 -17891.032} C_VEL
LIN {X 0,Y 269.44,Z 594.679,A -85,B 0,C 180,E1 -17893.327,E2 -17893.327} C_VEL
LIN {X 0,Y 268.956,Z 596.247,A -85,B 0,C 180,E1 -17895.206,E2 -17895.206} C_VEL
LIN {X 0,Y 268.402,Z 597.432,A -85,B 0,C 180,E1 -17897.909,E2 -17897.909} C_VEL
LIN {X 0,Y 268.196,Z 597.198,A -85,B 0,C 180,E1 -17900.954,E2 -17900.954} C_VEL
LIN {X 0,Y 268.258,Z 596.499,A -85,B 0,C 180,E1 -17902.473,E2 -17902.473} C_VEL
LIN {X 0,Y 268.448,Z 595.21,A -85,B 0,C 180,E1 -17904.187,E2 -17904.187} C_VEL
LIN {X 0,Y 268.661,Z 591.916,A -85,B 0,C 180,E1 -17907.001,E2 -17907.001} C_VEL
LIN {X 0,Y 269.16,Z 588.143,A -85,B 0,C 180,E1 -17909.252,E2 -17909.252} C_VEL
LIN {X 0,Y 269.779,Z 583.266,A -85,B 0,C 180,E1 -17911.493,E2 -17911.493} C_VEL
LIN {X 0,Y 270.762,Z 577.122,A -85,B 0,C 180,E1 -17913.721,E2 -17913.721} C_VEL
LIN {X 0,Y 272.01,Z 569.475,A -85,B 0,C 180,E1 -17915.932,E2 -17915.932} C_VEL
LIN {X 0,Y 273.518,Z 559.886,A -85,B 0,C 180,E1 -17918.124,E2 -17918.124} C_VEL
LIN {X 0,Y 275.061,Z 549.984,A -85,B 0,C 180,E1 -17919.931,E2 -17919.931} C_VEL
LIN {X 0,Y 276.604,Z 538.796,A -85,B 0,C 180,E1 -17921.542,E2 -17921.542} C_VEL
LIN {X 0,Y 277.814,Z 527.87,A -85,B 0,C 180,E1 -17922.788,E2 -17922.788} C_VEL
LIN {X 0,Y 278.859,Z 516.887,A -85,B 0,C 180,E1 -17923.759,E2 -17923.759} C_VEL
LIN {X 0,Y 279.793,Z 504.012,A -85,B 0,C 180,E1 -17924.593,E2 -17924.593} C_VEL
LIN {X 0,Y 280.337,Z 491.452,A -85,B 0,C 180,E1 -17925.117,E2 -17925.117} C_VEL
LIN {X 0,Y 282.227,Z 419,A -85,B 0,C 180,E1 -17926.941,E2 -17926.941} C_VEL
LIN {X 0,Y 275.436,Z 400.278,A -85,B 0,C 180,E1 -17928.058,E2 -17928.058} C_VEL
LIN {X 0,Y 271.394,Z 390.779,A -85,B 0,C 180,E1 -17928.706,E2 -17928.706} C_VEL
LIN {X 0,Y 270.314,Z 387.815,A -85,B 0,C 180,E1 -17928.896,E2 -17928.896} C_VEL
LIN {X 0,Y 270.236,Z 387.823,A -85,B 0,C 180,E1 -17932.96,E2 -17932.96} C_VEL
LIN {X 0,Y 270.274,Z 387.813,A -85,B 0,C 180,E1 -17936.234,E2 -17936.234} C_VEL
LIN {X 0,Y 270.239,Z 387.82,A -85,B 0,C 180,E1 -17939.611,E2 -17939.611} C_VEL
LIN {X 0,Y 270.217,Z 387.824,A -85,B 0,C 180,E1 -17943.665,E2 -17943.665} C_VEL
LIN {X 0,Y 270.22,Z 387.825,A -85,B 0,C 180,E1 -17946.74,E2 -17946.74} C_VEL
LIN {X 0,Y 270.173,Z 387.823,A -85,B 0,C 180,E1 -17951.028,E2 -17951.028} C_VEL
LIN {X 0,Y 270.188,Z 387.828,A -85,B 0,C 180,E1 -17954.611,E2 -17954.611} C_VEL
LIN {X 0,Y 270.266,Z 387.815,A -85,B 0,C 180,E1 -17958.947,E2 -17958.947} C_VEL
LIN {X 0,Y 270.241,Z 387.817,A -85,B 0,C 180,E1 -17963.262,E2 -17963.262} C_VEL
LIN {X 0,Y 270.201,Z 387.823,A -85,B 0,C 180,E1 -17966.892,E2 -17966.892} C_VEL
LIN {X 0,Y 270.192,Z 387.829,A -85,B 0,C 180,E1 -17970.382,E2 -17970.382} C_VEL
LIN {X 0,Y 270.258,Z 387.812,A -85,B 0,C 180,E1 -17973.763,E2 -17973.763} C_VEL
LIN {X 0,Y 270.233,Z 387.819,A -85,B 0,C 180,E1 -17977.038,E2 -17977.038} C_VEL
LIN {X 0,Y 270.299,Z 387.816,A -85,B 0,C 180,E1 -17980.244,E2 -17980.244} C_VEL
LIN {X 0,Y 270.392,Z 387.791,A -85,B 0,C 180,E1 -17984.934,E2 -17984.934} C_VEL
LIN {X 0,Y 270.436,Z 387.796,A -85,B 0,C 180,E1 -17989.508,E2 -17989.508} C_VEL
LIN {X 0,Y 270.172,Z 387.833,A -85,B 0,C 180,E1 -17990.341,E2 -17990.341} C_VEL
LIN {X 0,Y 268.834,Z 387.998,A -85,B 0,C 180,E1 -17991.57,E2 -17991.57} C_VEL
LIN {X 0,Y 264.462,Z 388.527,A -85,B 0,C 180,E1 -17994.43,E2 -17994.43} C_VEL
LIN {X 0,Y 263.478,Z 388.649,A -85,B 0,C 180,E1 -17995.71,E2 -17995.71} C_VEL
LIN {X 0,Y 263.439,Z 388.654,A -85,B 0,C 180,E1 -17996.144,E2 -17996.144} C_VEL
LIN {X 0,Y 263.747,Z 388.63,A -85,B 0,C 180,E1 -17998.473,E2 -17998.473} C_VEL
LIN {X 0,Y 263.747,Z 388.63,A -85,B 0,C 180,E1 -18001.527,E2 -18001.527} C_VEL
LIN {X 0,Y 263.567,Z 388.653,A -85,B 0,C 180,E1 -18007.661,E2 -18007.661} C_VEL
LIN {X 0,Y 263.369,Z 388.677,A -85,B 0,C 180,E1 -18010.765,E2 -18010.765} C_VEL
LIN {X 0,Y 263.339,Z 388.68,A -85,B 0,C 180,E1 -18015.478,E2 -18015.478} C_VEL
LIN {X 0,Y 263.264,Z 388.693,A -85,B 0,C 180,E1 -18020.306,E2 -18020.306} C_VEL
LIN {X 0,Y 263.203,Z 388.698,A -85,B 0,C 180,E1 -18025.292,E2 -18025.292} C_VEL
LIN {X 0,Y 263.161,Z 388.703,A -85,B 0,C 180,E1 -18028.732,E2 -18028.732} C_VEL
LIN {X 0,Y 263.128,Z 388.71,A -85,B 0,C 180,E1 -18032.289,E2 -18032.289} C_VEL
LIN {X 0,Y 263.186,Z 388.704,A -85,B 0,C 180,E1 -18035.978,E2 -18035.978} C_VEL
LIN {X 0,Y 263.157,Z 388.707,A -85,B 0,C 180,E1 -18039.863,E2 -18039.863} C_VEL
LIN {X 0,Y 263.142,Z 388.708,A -85,B 0,C 180,E1 -18043.98,E2 -18043.98} C_VEL
LIN {X 0,Y 263.149,Z 388.707,A -85,B 0,C 180,E1 -18048.4,E2 -18048.4} C_VEL
LIN {X 0,Y 263.165,Z 388.705,A -85,B 0,C 180,E1 -18052.105,E2 -18052.105} C_VEL
LIN {X 0,Y 263.235,Z 388.774,A -85,B 0,C 180,E1 -18054.594,E2 -18054.594} C_VEL
LIN {X 0,Y 265.885,Z 400.991,A -85,B 0,C 180,E1 -18058.974,E2 -18058.974} C_VEL
LIN {X 0,Y 267.578,Z 409.564,A -85,B 0,C 180,E1 -18061.828,E2 -18061.828} C_VEL
LIN {X 0,Y 269.187,Z 414.997,A -85,B 0,C 180,E1 -18062.138,E2 -18062.138} C_VEL
LIN {X 0,Y 273.578,Z 448.36,A -85,B 0,C 180,E1 -18063.483,E2 -18063.483} C_VEL
LIN {X 0,Y 274.844,Z 460.226,A -85,B 0,C 180,E1 -18063.922,E2 -18063.922} C_VEL
LIN {X 0,Y 273.187,Z 518.504,A -85,B 0,C 180,E1 -18065.445,E2 -18065.445} C_VEL
LIN {X 0,Y 272.327,Z 531.619,A -85,B 0,C 180,E1 -18066.068,E2 -18066.068} C_VEL
LIN {X 0,Y 271.125,Z 543.748,A -85,B 0,C 180,E1 -18066.918,E2 -18066.918} C_VEL
LIN {X 0,Y 269.751,Z 555.191,A -85,B 0,C 180,E1 -18068.006,E2 -18068.006} C_VEL
LIN {X 0,Y 268.054,Z 566.958,A -85,B 0,C 180,E1 -18069.472,E2 -18069.472} C_VEL
LIN {X 0,Y 266.384,Z 577.533,A -85,B 0,C 180,E1 -18071.144,E2 -18071.144} C_VEL
LIN {X 0,Y 265.034,Z 587.071,A -85,B 0,C 180,E1 -18073.041,E2 -18073.041} C_VEL
LIN {X 0,Y 263.613,Z 596.241,A -85,B 0,C 180,E1 -18075.329,E2 -18075.329} C_VEL
LIN {X 0,Y 262.419,Z 603.612,A -85,B 0,C 180,E1 -18077.629,E2 -18077.629} C_VEL
LIN {X 0,Y 261.737,Z 609.523,A -85,B 0,C 180,E1 -18079.949,E2 -18079.949} C_VEL
LIN {X 0,Y 261.339,Z 614.165,A -85,B 0,C 180,E1 -18082.273,E2 -18082.273} C_VEL
LIN {X 0,Y 261.179,Z 617.738,A -85,B 0,C 180,E1 -18084.637,E2 -18084.637} C_VEL
LIN {X 0,Y 261.221,Z 620.179,A -85,B 0,C 180,E1 -18086.916,E2 -18086.916} C_VEL
LIN {X 0,Y 261.228,Z 621.309,A -85,B 0,C 180,E1 -18088.458,E2 -18088.458} C_VEL
LIN {X 0,Y 261.248,Z 622.008,A -85,B 0,C 180,E1 -18090,E2 -18090} C_VEL
LIN {X 0,Y 261.197,Z 622.31,A -85,B 0,C 180,E1 -18091.542,E2 -18091.542} C_VEL
LIN {X 0,Y 261.166,Z 622.224,A -85,B 0,C 180,E1 -18093.085,E2 -18093.085} C_VEL
LIN {X 0,Y 261.131,Z 621.399,A -85,B 0,C 180,E1 -18095.249,E2 -18095.249} C_VEL
LIN {X 0,Y 261.321,Z 619.507,A -85,B 0,C 180,E1 -18097.728,E2 -18097.728} C_VEL
LIN {X 0,Y 261.85,Z 616.768,A -85,B 0,C 180,E1 -18100.047,E2 -18100.047} C_VEL
LIN {X 0,Y 262.658,Z 613.026,A -85,B 0,C 180,E1 -18102.36,E2 -18102.36} C_VEL
LIN {X 0,Y 264.007,Z 608.192,A -85,B 0,C 180,E1 -18104.648,E2 -18104.648} C_VEL
LIN {X 0,Y 265.692,Z 602.118,A -85,B 0,C 180,E1 -18106.916,E2 -18106.916} C_VEL
LIN {X 0,Y 267.503,Z 595.352,A -85,B 0,C 180,E1 -18108.948,E2 -18108.948} C_VEL
LIN {X 0,Y 269.709,Z 586.933,A -85,B 0,C 180,E1 -18110.995,E2 -18110.995} C_VEL
LIN {X 0,Y 272.189,Z 577.654,A -85,B 0,C 180,E1 -18112.786,E2 -18112.786} C_VEL
LIN {X 0,Y 274.578,Z 567.357,A -85,B 0,C 180,E1 -18114.376,E2 -18114.376} C_VEL
LIN {X 0,Y 276.984,Z 555.954,A -85,B 0,C 180,E1 -18115.754,E2 -18115.754} C_VEL
LIN {X 0,Y 279.071,Z 544.077,A -85,B 0,C 180,E1 -18116.854,E2 -18116.854} C_VEL
LIN {X 0,Y 280.746,Z 531.685,A -85,B 0,C 180,E1 -18117.689,E2 -18117.689} C_VEL
LIN {X 0,Y 281.981,Z 518.169,A -85,B 0,C 180,E1 -18118.303,E2 -18118.303} C_VEL
LIN {X 0,Y 284.141,Z 462.964,A -85,B 0,C 180,E1 -18119.708,E2 -18119.708} C_VEL
LIN {X 0,Y 281.227,Z 443.444,A -85,B 0,C 180,E1 -18120.683,E2 -18120.683} C_VEL
LIN {X 0,Y 278.687,Z 430.637,A -85,B 0,C 180,E1 -18121.43,E2 -18121.43} C_VEL
LIN {X 0,Y 272.139,Z 416.445,A -85,B 0,C 180,E1 -18122.847,E2 -18122.847} C_VEL
LIN {X 0,Y 268.123,Z 408.174,A -85,B 0,C 180,E1 -18123.758,E2 -18123.758} C_VEL
LIN {X 0,Y 265.935,Z 398.848,A -85,B 0,C 180,E1 -18127.55,E2 -18127.55} C_VEL
LIN {X 0,Y 263.697,Z 390.713,A -85,B 0,C 180,E1 -18131.157,E2 -18131.157} C_VEL
LIN {X 0,Y 263.133,Z 388.703,A -85,B 0,C 180,E1 -18132.148,E2 -18132.148} C_VEL
LIN {X 0,Y 263.144,Z 388.701,A -85,B 0,C 180,E1 -18136.145,E2 -18136.145} C_VEL
LIN {X 0,Y 263.157,Z 388.7,A -85,B 0,C 180,E1 -18140.137,E2 -18140.137} C_VEL
LIN {X 0,Y 263.186,Z 388.698,A -85,B 0,C 180,E1 -18144.022,E2 -18144.022} C_VEL
LIN {X 0,Y 263.129,Z 388.708,A -85,B 0,C 180,E1 -18147.711,E2 -18147.711} C_VEL
LIN {X 0,Y 263.197,Z 388.7,A -85,B 0,C 180,E1 -18151.783,E2 -18151.783} C_VEL
LIN {X 0,Y 263.221,Z 388.665,A -85,B 0,C 180,E1 -18155.2,E2 -18155.2} C_VEL
LIN {X 0,Y 263.258,Z 388.688,A -85,B 0,C 180,E1 -18159.693,E2 -18159.693} C_VEL
LIN {X 0,Y 263.339,Z 388.675,A -85,B 0,C 180,E1 -18164.522,E2 -18164.522} C_VEL
LIN {X 0,Y 263.369,Z 388.669,A -85,B 0,C 180,E1 -18169.235,E2 -18169.235} C_VEL
LIN {X 0,Y 263.566,Z 388.654,A -85,B 0,C 180,E1 -18172.339,E2 -18172.339} C_VEL
LIN {X 0,Y 263.747,Z 388.622,A -85,B 0,C 180,E1 -18178.473,E2 -18178.473} C_VEL
LIN {X 0,Y 263.746,Z 388.631,A -85,B 0,C 180,E1 -18181.527,E2 -18181.527} C_VEL
LIN {X 0,Y 263.553,Z 388.647,A -85,B 0,C 180,E1 -18187.663,E2 -18187.663} C_VEL
LIN {X 0,Y 263.35,Z 388.681,A -85,B 0,C 180,E1 -18190.767,E2 -18190.767} C_VEL
LIN {X 0,Y 263.34,Z 388.681,A -85,B 0,C 180,E1 -18195.479,E2 -18195.479} C_VEL
LIN {X 0,Y 263.259,Z 388.687,A -85,B 0,C 180,E1 -18200.307,E2 -18200.307} C_VEL
LIN {X 0,Y 263.204,Z 388.676,A -85,B 0,C 180,E1 -18205.292,E2 -18205.292} C_VEL
LIN {X 0,Y 263.176,Z 388.696,A -85,B 0,C 180,E1 -18208.731,E2 -18208.731} C_VEL
LIN {X 0,Y 263.131,Z 388.707,A -85,B 0,C 180,E1 -18212.289,E2 -18212.289} C_VEL
LIN {X 0,Y 263.188,Z 388.702,A -85,B 0,C 180,E1 -18215.979,E2 -18215.979} C_VEL
LIN {X 0,Y 263.16,Z 388.707,A -85,B 0,C 180,E1 -18219.863,E2 -18219.863} C_VEL
LIN {X 0,Y 263.205,Z 388.692,A -85,B 0,C 180,E1 -18221.878,E2 -18221.878} C_VEL
LIN {X 0,Y 263.195,Z 388.892,A -85,B 0,C 180,E1 -18226.412,E2 -18226.412} C_VEL
LIN {X 0,Y 264.37,Z 391.873,A -85,B 0,C 180,E1 -18226.767,E2 -18226.767} C_VEL
LIN {X 0,Y 265.925,Z 393.991,A -85,B 0,C 180,E1 -18227.103,E2 -18227.103} C_VEL
LIN {X 0,Y 270.836,Z 402.261,A -85,B 0,C 180,E1 -18228.18,E2 -18228.18} C_VEL
LIN {X 0,Y 279.14,Z 418.203,A -85,B 0,C 180,E1 -18229.94,E2 -18229.94} C_VEL
LIN {X 0,Y 285.095,Z 431.557,A -85,B 0,C 180,E1 -18231.175,E2 -18231.175} C_VEL
LIN {X 0,Y 282.763,Z 495.09,A -85,B 0,C 180,E1 -18232.799,E2 -18232.799} C_VEL
LIN {X 0,Y 281.813,Z 507.224,A -85,B 0,C 180,E1 -18233.348,E2 -18233.348} C_VEL
LIN {X 0,Y 280.364,Z 520.365,A -85,B 0,C 180,E1 -18234.242,E2 -18234.242} C_VEL
LIN {X 0,Y 278.302,Z 532.694,A -85,B 0,C 180,E1 -18235.376,E2 -18235.376} C_VEL
LIN {X 0,Y 276.32,Z 544.142,A -85,B 0,C 180,E1 -18236.81,E2 -18236.81} C_VEL
LIN {X 0,Y 274.259,Z 553.764,A -85,B 0,C 180,E1 -18238.311,E2 -18238.311} C_VEL
LIN {X 0,Y 271.868,Z 563.325,A -85,B 0,C 180,E1 -18240.158,E2 -18240.158} C_VEL
LIN {X 0,Y 269.769,Z 571.106,A -85,B 0,C 180,E1 -18242.036,E2 -18242.036} C_VEL
LIN {X 0,Y 267.617,Z 578.682,A -85,B 0,C 180,E1 -18244.323,E2 -18244.323} C_VEL
LIN {X 0,Y 265.708,Z 584.724,A -85,B 0,C 180,E1 -18246.625,E2 -18246.625} C_VEL
LIN {X 0,Y 264.13,Z 589.71,A -85,B 0,C 180,E1 -18249.089,E2 -18249.089} C_VEL
LIN {X 0,Y 263.053,Z 593.055,A -85,B 0,C 180,E1 -18251.301,E2 -18251.301} C_VEL
LIN {X 0,Y 262.49,Z 594.877,A -85,B 0,C 180,E1 -18252.872,E2 -18252.872} C_VEL
LIN {X 0,Y 261.914,Z 596.63,A -85,B 0,C 180,E1 -18255.018,E2 -18255.018} C_VEL
LIN {X 0,Y 261.363,Z 597.73,A -85,B 0,C 180,E1 -18257.578,E2 -18257.578} C_VEL
LIN {X 0,Y 261.152,Z 597.865,A -85,B 0,C 180,E1 -18259.142,E2 -18259.142} C_VEL
LIN {X 0,Y 261.159,Z 596.912,A -85,B 0,C 180,E1 -18262.267,E2 -18262.267} C_VEL
LIN {X 0,Y 261.356,Z 595.478,A -85,B 0,C 180,E1 -18264.247,E2 -18264.247} C_VEL
LIN {X 0,Y 261.567,Z 592.454,A -85,B 0,C 180,E1 -18266.92,E2 -18266.92} C_VEL
LIN {X 0,Y 262.075,Z 588.748,A -85,B 0,C 180,E1 -18269.232,E2 -18269.232} C_VEL
LIN {X 0,Y 262.713,Z 583.943,A -85,B 0,C 180,E1 -18271.533,E2 -18271.533} C_VEL
LIN {X 0,Y 263.708,Z 577.879,A -85,B 0,C 180,E1 -18273.82,E2 -18273.82} C_VEL
LIN {X 0,Y 264.977,Z 570.349,A -85,B 0,C 180,E1 -18276.09,E2 -18276.09} C_VEL
LIN {X 0,Y 266.267,Z 562.65,A -85,B 0,C 180,E1 -18277.965,E2 -18277.965} C_VEL
LIN {X 0,Y 267.926,Z 552.193,A -85,B 0,C 180,E1 -18280.008,E2 -18280.008} C_VEL
LIN {X 0,Y 269.499,Z 541.548,A -85,B 0,C 180,E1 -18281.66,E2 -18281.66} C_VEL
LIN {X 0,Y 270.809,Z 531.246,A -85,B 0,C 180,E1 -18282.934,E2 -18282.934} C_VEL
LIN {X 0,Y 272.01,Z 518.932,A -85,B 0,C 180,E1 -18284.113,E2 -18284.113} C_VEL
LIN {X 0,Y 273.067,Z 505.935,A -85,B 0,C 180,E1 -18285.009,E2 -18285.009} C_VEL
LIN {X 0,Y 273.657,Z 493.19,A -85,B 0,C 180,E1 -18285.596,E2 -18285.596} C_VEL
LIN {X 0,Y 275.665,Z 420.511,A -85,B 0,C 180,E1 -18287.471,E2 -18287.471} C_VEL
LIN {X 0,Y 268.781,Z 401.528,A -85,B 0,C 180,E1 -18288.648,E2 -18288.648} C_VEL
LIN {X 0,Y 264.298,Z 391.596,A -85,B 0,C 180,E1 -18289.382,E2 -18289.382} C_VEL
LIN {X 0,Y 263.26,Z 388.693,A -85,B 0,C 180,E1 -18289.592,E2 -18289.592} C_VEL
LIN {X 0,Y 263.23,Z 388.688,A -85,B 0,C 180,E1 -18294.799,E2 -18294.799} C_VEL
LIN {X 0,Y 263.187,Z 388.7,A -85,B 0,C 180,E1 -18298.728,E2 -18298.728} C_VEL
LIN {X 0,Y 263.135,Z 388.71,A -85,B 0,C 180,E1 -18302.287,E2 -18302.287} C_VEL
LIN {X 0,Y 263.165,Z 388.704,A -85,B 0,C 180,E1 -18305.981,E2 -18305.981} C_VEL
LIN {X 0,Y 263.108,Z 388.709,A -85,B 0,C 180,E1 -18309.871,E2 -18309.871} C_VEL
LIN {X 0,Y 263.138,Z 388.706,A -85,B 0,C 180,E1 -18313.98,E2 -18313.98} C_VEL
LIN {X 0,Y 263.209,Z 388.691,A -85,B 0,C 180,E1 -18318.384,E2 -18318.384} C_VEL
LIN {X 0,Y 263.205,Z 388.693,A -85,B 0,C 180,E1 -18323.229,E2 -18323.229} C_VEL
LIN {X 0,Y 263.182,Z 388.689,A -85,B 0,C 180,E1 -18325.889,E2 -18325.889} C_VEL
LIN {X 0,Y 263.138,Z 388.706,A -85,B 0,C 180,E1 -18329.505,E2 -18329.505} C_VEL
LIN {X 0,Y 263.188,Z 388.692,A -85,B 0,C 180,E1 -18333.001,E2 -18333.001} C_VEL
LIN {X 0,Y 263.183,Z 388.697,A -85,B 0,C 180,E1 -18336.386,E2 -18336.386} C_VEL
LIN {X 0,Y 263.265,Z 388.69,A -85,B 0,C 180,E1 -18339.693,E2 -18339.693} C_VEL
LIN {X 0,Y 263.34,Z 388.669,A -85,B 0,C 180,E1 -18344.521,E2 -18344.521} C_VEL
LIN {X 0,Y 263.389,Z 388.672,A -85,B 0,C 180,E1 -18349.534,E2 -18349.534} C_VEL
LIN {X 0,Y 263.567,Z 388.648,A -85,B 0,C 180,E1 -18352.338,E2 -18352.338} C_VEL
LIN {X 0,Y 263.439,Z 388.654,A -85,B 0,C 180,E1 -18356.144,E2 -18356.144} C_VEL
LIN {X 0,Y 262.905,Z 388.729,A -85,B 0,C 180,E1 -18357.422,E2 -18357.422} C_VEL
LIN {X 0,Y 260.165,Z 389.075,A -85,B 0,C 180,E1 -18359.509,E2 -18359.509} C_VEL
LIN {X 0,Y 256.884,Z 389.485,A -85,B 0,C 180,E1 -18362.078,E2 -18362.078} C_VEL
LIN {X 0,Y 256.509,Z 389.526,A -85,B 0,C 180,E1 -18362.967,E2 -18362.967} C_VEL
LIN {X 0,Y 256.534,Z 389.529,A -85,B 0,C 180,E1 -18367.873,E2 -18367.873} C_VEL
LIN {X 0,Y 256.304,Z 389.557,A -85,B 0,C 180,E1 -18371.066,E2 -18371.066} C_VEL
LIN {X 0,Y 256.289,Z 389.561,A -85,B 0,C 180,E1 -18375.915,E2 -18375.915} C_VEL
LIN {X 0,Y 256.213,Z 389.569,A -85,B 0,C 180,E1 -18380.891,E2 -18380.891} C_VEL
LIN {X 0,Y 256.183,Z 389.572,A -85,B 0,C 180,E1 -18385.139,E2 -18385.139} C_VEL
LIN {X 0,Y 256.099,Z 389.584,A -85,B 0,C 180,E1 -18389.601,E2 -18389.601} C_VEL
LIN {X 0,Y 256.081,Z 389.586,A -85,B 0,C 180,E1 -18393.291,E2 -18393.291} C_VEL
LIN {X 0,Y 256.137,Z 389.579,A -85,B 0,C 180,E1 -18397.279,E2 -18397.279} C_VEL
LIN {X 0,Y 256.1,Z 389.583,A -85,B 0,C 180,E1 -18401.194,E2 -18401.194} C_VEL
LIN {X 0,Y 256.07,Z 389.587,A -85,B 0,C 180,E1 -18405.527,E2 -18405.527} C_VEL
LIN {X 0,Y 256.079,Z 389.587,A -85,B 0,C 180,E1 -18408.802,E2 -18408.802} C_VEL
LIN {X 0,Y 256.143,Z 389.578,A -85,B 0,C 180,E1 -18412.871,E2 -18412.871} C_VEL
LIN {X 0,Y 256.216,Z 389.633,A -85,B 0,C 180,E1 -18414.044,E2 -18414.044} C_VEL
LIN {X 0,Y 258.822,Z 401.767,A -85,B 0,C 180,E1 -18418.538,E2 -18418.538} C_VEL
LIN {X 0,Y 260.268,Z 409.097,A -85,B 0,C 180,E1 -18421.087,E2 -18421.087} C_VEL
LIN {X 0,Y 262.804,Z 416.505,A -85,B 0,C 180,E1 -18421.564,E2 -18421.564} C_VEL
LIN {X 0,Y 267.023,Z 449.038,A -85,B 0,C 180,E1 -18422.914,E2 -18422.914} C_VEL
LIN {X 0,Y 268.276,Z 460.772,A -85,B 0,C 180,E1 -18423.364,E2 -18423.364} C_VEL
LIN {X 0,Y 266.581,Z 518.14,A -85,B 0,C 180,E1 -18424.897,E2 -18424.897} C_VEL
LIN {X 0,Y 265.69,Z 531.286,A -85,B 0,C 180,E1 -18425.536,E2 -18425.536} C_VEL
LIN {X 0,Y 264.437,Z 543.413,A -85,B 0,C 180,E1 -18426.402,E2 -18426.402} C_VEL
LIN {X 0,Y 262.908,Z 555.661,A -85,B 0,C 180,E1 -18427.609,E2 -18427.609} C_VEL
LIN {X 0,Y 261.171,Z 567.278,A -85,B 0,C 180,E1 -18429.112,E2 -18429.112} C_VEL
LIN {X 0,Y 259.454,Z 577.74,A -85,B 0,C 180,E1 -18430.826,E2 -18430.826} C_VEL
LIN {X 0,Y 258.089,Z 586.297,A -85,B 0,C 180,E1 -18432.57,E2 -18432.57} C_VEL
LIN {X 0,Y 257.133,Z 592.698,A -85,B 0,C 180,E1 -18434.138,E2 -18434.138} C_VEL
LIN {X 0,Y 255.854,Z 600.727,A -85,B 0,C 180,E1 -18436.498,E2 -18436.498} C_VEL
LIN {X 0,Y 254.936,Z 607.127,A -85,B 0,C 180,E1 -18438.874,E2 -18438.874} C_VEL
LIN {X 0,Y 254.405,Z 612.214,A -85,B 0,C 180,E1 -18441.261,E2 -18441.261} C_VEL
LIN {X 0,Y 254.15,Z 616.143,A -85,B 0,C 180,E1 -18443.65,E2 -18443.65} C_VEL
LIN {X 0,Y 254.071,Z 618.158,A -85,B 0,C 180,E1 -18445.24,E2 -18445.24} C_VEL
LIN {X 0,Y 254.129,Z 619.755,A -85,B 0,C 180,E1 -18446.829,E2 -18446.829} C_VEL
LIN {X 0,Y 254.153,Z 620.925,A -85,B 0,C 180,E1 -18448.415,E2 -18448.415} C_VEL
LIN {X 0,Y 254.17,Z 621.645,A -85,B 0,C 180,E1 -18450,E2 -18450} C_VEL
LIN {X 0,Y 254.122,Z 621.967,A -85,B 0,C 180,E1 -18451.585,E2 -18451.585} C_VEL
LIN {X 0,Y 254.075,Z 621.9,A -85,B 0,C 180,E1 -18453.171,E2 -18453.171} C_VEL
LIN {X 0,Y 254.053,Z 621.218,A -85,B 0,C 180,E1 -18455.199,E2 -18455.199} C_VEL
LIN {X 0,Y 254.262,Z 619.262,A -85,B 0,C 180,E1 -18457.944,E2 -18457.944} C_VEL
LIN {X 0,Y 254.818,Z 616.564,A -85,B 0,C 180,E1 -18460.327,E2 -18460.327} C_VEL
LIN {X 0,Y 255.688,Z 612.867,A -85,B 0,C 180,E1 -18462.702,E2 -18462.702} C_VEL
LIN {X 0,Y 257.124,Z 608.082,A -85,B 0,C 180,E1 -18465.05,E2 -18465.05} C_VEL
LIN {X 0,Y 258.884,Z 602.06,A -85,B 0,C 180,E1 -18467.374,E2 -18467.374} C_VEL
LIN {X 0,Y 260.989,Z 594.596,A -85,B 0,C 180,E1 -18469.669,E2 -18469.669} C_VEL
LIN {X 0,Y 263.082,Z 587.003,A -85,B 0,C 180,E1 -18471.55,E2 -18471.55} C_VEL
LIN {X 0,Y 265.673,Z 577.833,A -85,B 0,C 180,E1 -18473.378,E2 -18473.378} C_VEL
LIN {X 0,Y 268.149,Z 567.664,A -85,B 0,C 180,E1 -18475,E2 -18475} C_VEL
LIN {X 0,Y 270.637,Z 556.409,A -85,B 0,C 180,E1 -18476.404,E2 -18476.404} C_VEL
LIN {X 0,Y 272.623,Z 545.749,A -85,B 0,C 180,E1 -18477.438,E2 -18477.438} C_VEL
LIN {X 0,Y 274.499,Z 532.876,A -85,B 0,C 180,E1 -18478.375,E2 -18478.375} C_VEL
LIN {X 0,Y 275.806,Z 520.039,A -85,B 0,C 180,E1 -18479,E2 -18479} C_VEL
LIN {X 0,Y 276.722,Z 502.137,A -85,B 0,C 180,E1 -18479.513,E2 -18479.513} C_VEL
LIN {X 0,Y 278.138,Z 463.166,A -85,B 0,C 180,E1 -18480.508,E2 -18480.508} C_VEL
LIN {X 0,Y 274.555,Z 440.269,A -85,B 0,C 180,E1 -18481.728,E2 -18481.728} C_VEL
LIN {X 0,Y 273.051,Z 433.343,A -85,B 0,C 180,E1 -18482.169,E2 -18482.169} C_VEL
LIN {X 0,Y 265.345,Z 416.744,A -85,B 0,C 180,E1 -18483.919,E2 -18483.919} C_VEL
LIN {X 0,Y 260.779,Z 407.629,A -85,B 0,C 180,E1 -18485.044,E2 -18485.044} C_VEL
LIN {X 0,Y 259.054,Z 400.408,A -85,B 0,C 180,E1 -18488.117,E2 -18488.117} C_VEL
LIN {X 0,Y 257.062,Z 393.1,A -85,B 0,C 180,E1 -18491.468,E2 -18491.468} C_VEL
LIN {X 0,Y 256.105,Z 389.578,A -85,B 0,C 180,E1 -18493.24,E2 -18493.24} C_VEL
LIN {X 0,Y 256.122,Z 389.576,A -85,B 0,C 180,E1 -18497.805,E2 -18497.805} C_VEL
LIN {X 0,Y 256.105,Z 389.579,A -85,B 0,C 180,E1 -18500.864,E2 -18500.864} C_VEL
LIN {X 0,Y 256.117,Z 389.579,A -85,B 0,C 180,E1 -18504.813,E2 -18504.813} C_VEL
LIN {X 0,Y 256.088,Z 389.585,A -85,B 0,C 180,E1 -18508.572,E2 -18508.572} C_VEL
LIN {X 0,Y 256.137,Z 389.578,A -85,B 0,C 180,E1 -18512.196,E2 -18512.196} C_VEL
LIN {X 0,Y 256.162,Z 389.545,A -85,B 0,C 180,E1 -18515.699,E2 -18515.699} C_VEL
LIN {X 0,Y 256.162,Z 389.577,A -85,B 0,C 180,E1 -18519.105,E2 -18519.105} C_VEL
LIN {X 0,Y 256.289,Z 389.556,A -85,B 0,C 180,E1 -18524.085,E2 -18524.085} C_VEL
LIN {X 0,Y 256.304,Z 389.55,A -85,B 0,C 180,E1 -18528.934,E2 -18528.934} C_VEL
LIN {X 0,Y 256.534,Z 389.53,A -85,B 0,C 180,E1 -18532.127,E2 -18532.127} C_VEL
LIN {X 0,Y 256.709,Z 389.499,A -85,B 0,C 180,E1 -18538.432,E2 -18538.432} C_VEL
LIN {X 0,Y 256.709,Z 389.507,A -85,B 0,C 180,E1 -18541.569,E2 -18541.569} C_VEL
LIN {X 0,Y 256.466,Z 389.534,A -85,B 0,C 180,E1 -18546.743,E2 -18546.743} C_VEL
LIN {X 0,Y 256.422,Z 389.542,A -85,B 0,C 180,E1 -18549.466,E2 -18549.466} C_VEL
LIN {X 0,Y 256.246,Z 389.564,A -85,B 0,C 180,E1 -18554.291,E2 -18554.291} C_VEL
LIN {X 0,Y 256.2,Z 389.565,A -85,B 0,C 180,E1 -18557.563,E2 -18557.563} C_VEL
LIN {X 0,Y 256.153,Z 389.57,A -85,B 0,C 180,E1 -18561.12,E2 -18561.12} C_VEL
LIN {X 0,Y 256.185,Z 389.552,A -85,B 0,C 180,E1 -18565.139,E2 -18565.139} C_VEL
LIN {X 0,Y 256.111,Z 389.583,A -85,B 0,C 180,E1 -18569.601,E2 -18569.601} C_VEL
LIN {X 0,Y 256.083,Z 389.586,A -85,B 0,C 180,E1 -18573.291,E2 -18573.291} C_VEL
LIN {X 0,Y 256.139,Z 389.578,A -85,B 0,C 180,E1 -18577.28,E2 -18577.28} C_VEL
LIN {X 0,Y 256.13,Z 389.58,A -85,B 0,C 180,E1 -18581.19,E2 -18581.19} C_VEL
LIN {X 0,Y 256.06,Z 389.592,A -85,B 0,C 180,E1 -18585.196,E2 -18585.196} C_VEL
LIN {X 0,Y 257.097,Z 392.456,A -85,B 0,C 180,E1 -18585.495,E2 -18585.495} C_VEL
LIN {X 0,Y 258.986,Z 394.973,A -85,B 0,C 180,E1 -18585.928,E2 -18585.928} C_VEL
LIN {X 0,Y 264.597,Z 404.042,A -85,B 0,C 180,E1 -18587.218,E2 -18587.218} C_VEL
LIN {X 0,Y 271.891,Z 417.716,A -85,B 0,C 180,E1 -18588.845,E2 -18588.845} C_VEL
LIN {X 0,Y 278.46,Z 431.868,A -85,B 0,C 180,E1 -18590.264,E2 -18590.264} C_VEL
LIN {X 0,Y 279.227,Z 433.939,A -85,B 0,C 180,E1 -18590.437,E2 -18590.437} C_VEL
LIN {X 0,Y 276.738,Z 495.889,A -85,B 0,C 180,E1 -18592.043,E2 -18592.043} C_VEL
LIN {X 0,Y 275.784,Z 507.556,A -85,B 0,C 180,E1 -18592.583,E2 -18592.583} C_VEL
LIN {X 0,Y 274.36,Z 520.12,A -85,B 0,C 180,E1 -18593.448,E2 -18593.448} C_VEL
LIN {X 0,Y 272.359,Z 531.795,A -85,B 0,C 180,E1 -18594.509,E2 -18594.509} C_VEL
LIN {X 0,Y 270.37,Z 542.802,A -85,B 0,C 180,E1 -18595.866,E2 -18595.866} C_VEL
LIN {X 0,Y 268.132,Z 553.275,A -85,B 0,C 180,E1 -18597.499,E2 -18597.499} C_VEL
LIN {X 0,Y 265.571,Z 562.998,A -85,B 0,C 180,E1 -18599.375,E2 -18599.375} C_VEL
LIN {X 0,Y 263.366,Z 570.913,A -85,B 0,C 180,E1 -18601.293,E2 -18601.293} C_VEL
LIN {X 0,Y 261.073,Z 578.586,A -85,B 0,C 180,E1 -18603.63,E2 -18603.63} C_VEL
LIN {X 0,Y 259.05,Z 584.711,A -85,B 0,C 180,E1 -18605.987,E2 -18605.987} C_VEL
LIN {X 0,Y 257.585,Z 588.996,A -85,B 0,C 180,E1 -18608.075,E2 -18608.075} C_VEL
LIN {X 0,Y 256.175,Z 593.187,A -85,B 0,C 180,E1 -18610.78,E2 -18610.78} C_VEL
LIN {X 0,Y 255.548,Z 595.061,A -85,B 0,C 180,E1 -18612.391,E2 -18612.391} C_VEL
LIN {X 0,Y 254.863,Z 597.021,A -85,B 0,C 180,E1 -18614.831,E2 -18614.831} C_VEL
LIN {X 0,Y 254.34,Z 598.021,A -85,B 0,C 180,E1 -18617.229,E2 -18617.229} C_VEL
LIN {X 0,Y 254.087,Z 598.213,A -85,B 0,C 180,E1 -18618.836,E2 -18618.836} C_VEL
LIN {X 0,Y 254.025,Z 597.964,A -85,B 0,C 180,E1 -18620.445,E2 -18620.445} C_VEL
LIN {X 0,Y 254.202,Z 596.299,A -85,B 0,C 180,E1 -18623.651,E2 -18623.651} C_VEL
LIN {X 0,Y 254.318,Z 594.871,A -85,B 0,C 180,E1 -18625.245,E2 -18625.245} C_VEL
LIN {X 0,Y 254.59,Z 591.918,A -85,B 0,C 180,E1 -18627.627,E2 -18627.627} C_VEL
LIN {X 0,Y 255.162,Z 587.927,A -85,B 0,C 180,E1 -18630,E2 -18630} C_VEL
LIN {X 0,Y 256.046,Z 581.799,A -85,B 0,C 180,E1 -18632.753,E2 -18632.753} C_VEL
LIN {X 0,Y 257.241,Z 575.115,A -85,B 0,C 180,E1 -18635.094,E2 -18635.094} C_VEL
LIN {X 0,Y 258.727,Z 566.829,A -85,B 0,C 180,E1 -18637.413,E2 -18637.413} C_VEL
LIN {X 0,Y 260.148,Z 558.305,A -85,B 0,C 180,E1 -18639.328,E2 -18639.328} C_VEL
LIN {X 0,Y 261.899,Z 547.786,A -85,B 0,C 180,E1 -18641.218,E2 -18641.218} C_VEL
LIN {X 0,Y 263.419,Z 537.36,A -85,B 0,C 180,E1 -18642.715,E2 -18642.715} C_VEL
LIN {X 0,Y 264.693,Z 525.907,A -85,B 0,C 180,E1 -18644.021,E2 -18644.021} C_VEL
LIN {X 0,Y 265.873,Z 513.996,A -85,B 0,C 180,E1 -18645.033,E2 -18645.033} C_VEL
LIN {X 0,Y 266.714,Z 501.15,A -85,B 0,C 180,E1 -18645.816,E2 -18645.816} C_VEL
LIN {X 0,Y 267.27,Z 487.486,A -85,B 0,C 180,E1 -18646.321,E2 -18646.321} C_VEL
LIN {X 0,Y 269.127,Z 422.084,A -85,B 0,C 180,E1 -18648.024,E2 -18648.024} C_VEL
LIN {X 0,Y 262.732,Z 404.371,A -85,B 0,C 180,E1 -18649.163,E2 -18649.163} C_VEL
LIN {X 0,Y 256.997,Z 391.997,A -85,B 0,C 180,E1 -18650.133,E2 -18650.133} C_VEL
LIN {X 0,Y 256.243,Z 389.568,A -85,B 0,C 180,E1 -18650.309,E2 -18650.309} C_VEL
LIN {X 0,Y 256.193,Z 389.563,A -85,B 0,C 180,E1 -18655.138,E2 -18655.138} C_VEL
LIN {X 0,Y 256.119,Z 389.579,A -85,B 0,C 180,E1 -18659.598,E2 -18659.598} C_VEL
LIN {X 0,Y 256.078,Z 389.585,A -85,B 0,C 180,E1 -18663.29,E2 -18663.29} C_VEL
LIN {X 0,Y 256.117,Z 389.58,A -85,B 0,C 180,E1 -18667.27,E2 -18667.27} C_VEL
LIN {X 0,Y 256.059,Z 389.58,A -85,B 0,C 180,E1 -18671.201,E2 -18671.201} C_VEL
LIN {X 0,Y 256.075,Z 389.583,A -85,B 0,C 180,E1 -18675.525,E2 -18675.525} C_VEL
LIN {X 0,Y 256.13,Z 389.576,A -85,B 0,C 180,E1 -18678.81,E2 -18678.81} C_VEL
LIN {X 0,Y 256.154,Z 389.572,A -85,B 0,C 180,E1 -18682.871,E2 -18682.871} C_VEL
LIN {X 0,Y 256.083,Z 389.581,A -85,B 0,C 180,E1 -18686.709,E2 -18686.709} C_VEL
LIN {X 0,Y 256.123,Z 389.578,A -85,B 0,C 180,E1 -18691.409,E2 -18691.409} C_VEL
LIN {X 0,Y 256.165,Z 389.565,A -85,B 0,C 180,E1 -18695.698,E2 -18695.698} C_VEL
LIN {X 0,Y 256.215,Z 389.568,A -85,B 0,C 180,E1 -18699.108,E2 -18699.108} C_VEL
LIN {X 0,Y 256.29,Z 389.546,A -85,B 0,C 180,E1 -18704.084,E2 -18704.084} C_VEL
LIN {X 0,Y 256.305,Z 389.556,A -85,B 0,C 180,E1 -18708.933,E2 -18708.933} C_VEL
LIN {X 0,Y 256.534,Z 389.525,A -85,B 0,C 180,E1 -18712.126,E2 -18712.126} C_VEL
LIN {X 0,Y 256.709,Z 389.507,A -85,B 0,C 180,E1 -18718.431,E2 -18718.431} C_VEL
LIN {X 0,Y 256.71,Z 389.506,A -85,B 0,C 180,E1 -18721.568,E2 -18721.568} C_VEL
LIN {X 0,Y 256.509,Z 389.526,A -85,B 0,C 180,E1 -18722.967,E2 -18722.967} C_VEL
LIN {X 0,Y 255.79,Z 389.623,A -85,B 0,C 180,E1 -18724.276,E2 -18724.276} C_VEL
LIN {X 0,Y 252.982,Z 389.975,A -85,B 0,C 180,E1 -18726.414,E2 -18726.414} C_VEL
LIN {X 0,Y 249.748,Z 390.375,A -85,B 0,C 180,E1 -18729.044,E2 -18729.044} C_VEL
LIN {X 0,Y 249.354,Z 390.421,A -85,B 0,C 180,E1 -18729.954,E2 -18729.954} C_VEL
LIN {X 0,Y 249.196,Z 390.441,A -85,B 0,C 180,E1 -18734.704,E2 -18734.704} C_VEL
LIN {X 0,Y 249.135,Z 390.45,A -85,B 0,C 180,E1 -18738.077,E2 -18738.077} C_VEL
LIN {X 0,Y 249.099,Z 390.456,A -85,B 0,C 180,E1 -18741.517,E2 -18741.517} C_VEL
LIN {X 0,Y 249.126,Z 390.452,A -85,B 0,C 180,E1 -18745.482,E2 -18745.482} C_VEL
LIN {X 0,Y 249.068,Z 390.458,A -85,B 0,C 180,E1 -18748.989,E2 -18748.989} C_VEL
LIN {X 0,Y 249.032,Z 390.465,A -85,B 0,C 180,E1 -18752.425,E2 -18752.425} C_VEL
LIN {X 0,Y 249.072,Z 390.46,A -85,B 0,C 180,E1 -18756.338,E2 -18756.338} C_VEL
LIN {X 0,Y 249.074,Z 390.459,A -85,B 0,C 180,E1 -18760.464,E2 -18760.464} C_VEL
LIN {X 0,Y 249.017,Z 390.463,A -85,B 0,C 180,E1 -18764.876,E2 -18764.876} C_VEL
LIN {X 0,Y 249.03,Z 390.465,A -85,B 0,C 180,E1 -18767.367,E2 -18767.367} C_VEL
LIN {X 0,Y 249.04,Z 390.465,A -85,B 0,C 180,E1 -18771.623,E2 -18771.623} C_VEL
LIN {X 0,Y 249.14,Z 390.575,A -85,B 0,C 180,E1 -18773.486,E2 -18773.486} C_VEL
LIN {X 0,Y 251.342,Z 400.606,A -85,B 0,C 180,E1 -18777.356,E2 -18777.356} C_VEL
LIN {X 0,Y 252.957,Z 408.721,A -85,B 0,C 180,E1 -18780.303,E2 -18780.303} C_VEL
LIN {X 0,Y 256.542,Z 418.851,A -85,B 0,C 180,E1 -18780.996,E2 -18780.996} C_VEL
LIN {X 0,Y 260.581,Z 450.536,A -85,B 0,C 180,E1 -18782.352,E2 -18782.352} C_VEL
LIN {X 0,Y 261.713,Z 462.311,A -85,B 0,C 180,E1 -18782.807,E2 -18782.807} C_VEL
LIN {X 0,Y 259.97,Z 518.152,A -85,B 0,C 180,E1 -18784.336,E2 -18784.336} C_VEL
LIN {X 0,Y 259.006,Z 531.72,A -85,B 0,C 180,E1 -18785.022,E2 -18785.022} C_VEL
LIN {X 0,Y 257.674,Z 544.193,A -85,B 0,C 180,E1 -18785.958,E2 -18785.958} C_VEL
LIN {X 0,Y 256.096,Z 556.129,A -85,B 0,C 180,E1 -18787.193,E2 -18787.193} C_VEL
LIN {X 0,Y 254.298,Z 567.598,A -85,B 0,C 180,E1 -18788.732,E2 -18788.732} C_VEL
LIN {X 0,Y 252.539,Z 577.933,A -85,B 0,C 180,E1 -18790.492,E2 -18790.492} C_VEL
LIN {X 0,Y 251.041,Z 587.225,A -85,B 0,C 180,E1 -18792.486,E2 -18792.486} C_VEL
LIN {X 0,Y 249.731,Z 594.881,A -85,B 0,C 180,E1 -18794.494,E2 -18794.494} C_VEL
LIN {X 0,Y 248.477,Z 602.38,A -85,B 0,C 180,E1 -18796.923,E2 -18796.923} C_VEL
LIN {X 0,Y 247.699,Z 608.401,A -85,B 0,C 180,E1 -18799.373,E2 -18799.373} C_VEL
LIN {X 0,Y 247.218,Z 613.144,A -85,B 0,C 180,E1 -18801.828,E2 -18801.828} C_VEL
LIN {X 0,Y 246.989,Z 617.397,A -85,B 0,C 180,E1 -18804.818,E2 -18804.818} C_VEL
LIN {X 0,Y 247.039,Z 619.33,A -85,B 0,C 180,E1 -18806.738,E2 -18806.738} C_VEL
LIN {X 0,Y 247.079,Z 620.532,A -85,B 0,C 180,E1 -18808.37,E2 -18808.37} C_VEL
LIN {X 0,Y 247.094,Z 621.282,A -85,B 0,C 180,E1 -18810,E2 -18810} C_VEL
LIN {X 0,Y 247.048,Z 621.624,A -85,B 0,C 180,E1 -18811.63,E2 -18811.63} C_VEL
LIN {X 0,Y 246.987,Z 621.575,A -85,B 0,C 180,E1 -18813.262,E2 -18813.262} C_VEL
LIN {X 0,Y 246.943,Z 621.076,A -85,B 0,C 180,E1 -18815.063,E2 -18815.063} C_VEL
LIN {X 0,Y 247.202,Z 619.017,A -85,B 0,C 180,E1 -18818.172,E2 -18818.172} C_VEL
LIN {X 0,Y 247.806,Z 616.361,A -85,B 0,C 180,E1 -18820.623,E2 -18820.623} C_VEL
LIN {X 0,Y 248.728,Z 612.709,A -85,B 0,C 180,E1 -18823.064,E2 -18823.064} C_VEL
LIN {X 0,Y 250.258,Z 607.971,A -85,B 0,C 180,E1 -18825.473,E2 -18825.473} C_VEL
LIN {X 0,Y 252.47,Z 600.894,A -85,B 0,C 180,E1 -18828.246,E2 -18828.246} C_VEL
LIN {X 0,Y 254.7,Z 593.235,A -85,B 0,C 180,E1 -18830.597,E2 -18830.597} C_VEL
LIN {X 0,Y 256.992,Z 585.432,A -85,B 0,C 180,E1 -18832.51,E2 -18832.51} C_VEL
LIN {X 0,Y 260.006,Z 574.86,A -85,B 0,C 180,E1 -18834.556,E2 -18834.556} C_VEL
LIN {X 0,Y 262.674,Z 564.128,A -85,B 0,C 180,E1 -18836.197,E2 -18836.197} C_VEL
LIN {X 0,Y 264.909,Z 553.72,A -85,B 0,C 180,E1 -18837.448,E2 -18837.448} C_VEL
LIN {X 0,Y 267.246,Z 541.213,A -85,B 0,C 180,E1 -18838.573,E2 -18838.573} C_VEL
LIN {X 0,Y 269.084,Z 528.042,A -85,B 0,C 180,E1 -18839.429,E2 -18839.429} C_VEL
LIN {X 0,Y 270.19,Z 515.552,A -85,B 0,C 180,E1 -18839.963,E2 -18839.963} C_VEL
LIN {X 0,Y 272.254,Z 464.155,A -85,B 0,C 180,E1 -18841.311,E2 -18841.311} C_VEL
LIN {X 0,Y 268.513,Z 440.325,A -85,B 0,C 180,E1 -18842.635,E2 -18842.635} C_VEL
LIN {X 0,Y 267.404,Z 435.914,A -85,B 0,C 180,E1 -18842.952,E2 -18842.952} C_VEL
LIN {X 0,Y 259.825,Z 419.647,A -85,B 0,C 180,E1 -18844.753,E2 -18844.753} C_VEL
LIN {X 0,Y 255.183,Z 410.837,A -85,B 0,C 180,E1 -18845.891,E2 -18845.891} C_VEL
LIN {X 0,Y 253.554,Z 407.292,A -85,B 0,C 180,E1 -18846.335,E2 -18846.335} C_VEL
LIN {X 0,Y 251.476,Z 399.197,A -85,B 0,C 180,E1 -18849.998,E2 -18849.998} C_VEL
LIN {X 0,Y 249.039,Z 390.462,A -85,B 0,C 180,E1 -18854.329,E2 -18854.329} C_VEL
LIN {X 0,Y 249.059,Z 390.454,A -85,B 0,C 180,E1 -18857.372,E2 -18857.372} C_VEL
LIN {X 0,Y 249.049,Z 390.458,A -85,B 0,C 180,E1 -18861.624,E2 -18861.624} C_VEL
LIN {X 0,Y 249.058,Z 390.459,A -85,B 0,C 180,E1 -18865.642,E2 -18865.642} C_VEL
LIN {X 0,Y 249.047,Z 390.457,A -85,B 0,C 180,E1 -18869.473,E2 -18869.473} C_VEL
LIN {X 0,Y 249.069,Z 390.443,A -85,B 0,C 180,E1 -18873.162,E2 -18873.162} C_VEL
LIN {X 0,Y 249.074,Z 390.439,A -85,B 0,C 180,E1 -18876.732,E2 -18876.732} C_VEL
LIN {X 0,Y 249.105,Z 390.448,A -85,B 0,C 180,E1 -18880.211,E2 -18880.211} C_VEL
LIN {X 0,Y 249.237,Z 390.436,A -85,B 0,C 180,E1 -18883.622,E2 -18883.622} C_VEL
LIN {X 0,Y 249.248,Z 390.431,A -85,B 0,C 180,E1 -18888.617,E2 -18888.617} C_VEL
LIN {X 0,Y 249.476,Z 390.409,A -85,B 0,C 180,E1 -18891.903,E2 -18891.903} C_VEL
LIN {X 0,Y 249.432,Z 390.416,A -85,B 0,C 180,E1 -18896.77,E2 -18896.77} C_VEL
LIN {X 0,Y 249.73,Z 390.374,A -85,B 0,C 180,E1 -18900,E2 -18900} C_VEL
LIN {X 0,Y 249.43,Z 390.404,A -85,B 0,C 180,E1 -18903.231,E2 -18903.231} C_VEL
LIN {X 0,Y 249.435,Z 390.41,A -85,B 0,C 180,E1 -18906.728,E2 -18906.728} C_VEL
LIN {X 0,Y 249.339,Z 390.425,A -85,B 0,C 180,E1 -18909.737,E2 -18909.737} C_VEL
LIN {X 0,Y 249.193,Z 390.446,A -85,B 0,C 180,E1 -18914.705,E2 -18914.705} C_VEL
LIN {X 0,Y 249.131,Z 390.448,A -85,B 0,C 180,E1 -18918.078,E2 -18918.078} C_VEL
LIN {X 0,Y 249.084,Z 390.451,A -85,B 0,C 180,E1 -18921.519,E2 -18921.519} C_VEL
LIN {X 0,Y 249.127,Z 390.426,A -85,B 0,C 180,E1 -18925.483,E2 -18925.483} C_VEL
LIN {X 0,Y 249.08,Z 390.455,A -85,B 0,C 180,E1 -18928.994,E2 -18928.994} C_VEL
LIN {X 0,Y 249.034,Z 390.464,A -85,B 0,C 180,E1 -18932.426,E2 -18932.426} C_VEL
LIN {X 0,Y 249.074,Z 390.458,A -85,B 0,C 180,E1 -18936.339,E2 -18936.339} C_VEL
LIN {X 0,Y 249.082,Z 390.464,A -85,B 0,C 180,E1 -18940.464,E2 -18940.464} C_VEL
LIN {X 0,Y 249.051,Z 390.534,A -85,B 0,C 180,E1 -18943.869,E2 -18943.869} C_VEL
LIN {X 0,Y 250.019,Z 393.297,A -85,B 0,C 180,E1 -18944.167,E2 -18944.167} C_VEL
LIN {X 0,Y 251.985,Z 395.902,A -85,B 0,C 180,E1 -18944.651,E2 -18944.651} C_VEL
LIN {X 0,Y 259.361,Z 407.412,A -85,B 0,C 180,E1 -18946.43,E2 -18946.43} C_VEL
LIN {X 0,Y 267.134,Z 422.246,A -85,B 0,C 180,E1 -18948.244,E2 -18948.244} C_VEL
LIN {X 0,Y 273.254,Z 435.553,A -85,B 0,C 180,E1 -18949.621,E2 -18949.621} C_VEL
LIN {X 0,Y 270.848,Z 495.408,A -85,B 0,C 180,E1 -18951.201,E2 -18951.201} C_VEL
LIN {X 0,Y 269.808,Z 507.895,A -85,B 0,C 180,E1 -18951.784,E2 -18951.784} C_VEL
LIN {X 0,Y 268.253,Z 521.036,A -85,B 0,C 180,E1 -18952.711,E2 -18952.711} C_VEL
LIN {X 0,Y 266.167,Z 532.551,A -85,B 0,C 180,E1 -18953.787,E2 -18953.787} C_VEL
LIN {X 0,Y 264.193,Z 543.073,A -85,B 0,C 180,E1 -18955.115,E2 -18955.115} C_VEL
LIN {X 0,Y 261.699,Z 554.111,A -85,B 0,C 180,E1 -18956.876,E2 -18956.876} C_VEL
LIN {X 0,Y 259.349,Z 562.656,A -85,B 0,C 180,E1 -18958.558,E2 -18958.558} C_VEL
LIN {X 0,Y 257.018,Z 570.696,A -85,B 0,C 180,E1 -18960.516,E2 -18960.516} C_VEL
LIN {X 0,Y 254.585,Z 578.496,A -85,B 0,C 180,E1 -18962.904,E2 -18962.904} C_VEL
